(*=====================================================================*)
	IF 	Service.daten[i].Type_Service = STUNDEN THEN
		Service.visu[i].BtnType.Text := 'TIMER';
		Service.visu[i].BtnType.Pressed := FALSE;
	ELSIF 	Service.daten[i].Type_Service = TAGE THEN
		Service.visu[i].BtnType.Text := 'TIMER';
		Service.visu[i].BtnType.Pressed := FALSE;
	ELSIF Service.daten[i].Type_Service = COUNTER THEN
		Service.visu[i].BtnType.Text := 'COUNT';
		Service.visu[i].BtnType.Pressed := TRUE;
	END_IF
	Service.visu[i].BtnType.Enable := TRUE;
	Service.visu[i].BtnType.BackgroundColor := Color.lightgrey;
	Service.visu[i].BtnType.TextColor := Color.black;
	Service.visu[i].BtnType.Visible := TRUE;
END_FOR
END_ACTION
ACTION Reset:
k:=-1;
FOR k:=1 TO 3 BY 1 DO
	IF	gVarSystemtime.wHour >(MP.ShiftData.Shift[k].TimeStart.wHour + 1) AND NOT Reset_Help[k] THEN
		i:=-1;
		FOR i:=0 TO 15 BY 1 DO
			Default_reached[i] := FALSE;
		END_FOR
		Reset_Help[k]:=TRUE;
	END_IF
END_FOR

IF	gVarSystemtime.wHour < MP.ShiftData.Shift[1].TimeStart.wHour THEN
	k:=-1;
	FOR k:=1 TO 3 BY 1 DO
		Reset_Help[k]:=FALSE;
	END_FOR
END_IF
END_ACTION
ACTION Umschalten:
i := -1;

FOR i:=0 TO 15 BY 1 DO

(* Umschaltung der Funktion (Zeit oder Stückzahl) *)
	IF NOT b_first_cycle THEN
		IF	M_BtnType[i] AND NOT Service.visu[i].BtnType.Pressed THEN
				Service.daten[i].Starttag := 0;
				Service.daten[i].Startstunden := 0;
				Service.daten[i].StartBetriebsStd := 0;
				Service.daten[i].Current_Value := 0;
				IF	Service.daten[i].Type_Service < COUNTER THEN
						Service.daten[i].Type_Service:=Service.daten[i].Type_Service+1;
				ELSE
						Service.daten[i].Type_Service:=0;
				END_IF
		END_IF
		M_BtnType[i]:=Service.visu[i].BtnType.Pressed;

		IF	Service.daten[i].Type_Service = BETRIEBSSTUNDEN THEN
				Service.visu[i].BtnType.Text := 'TIMER';
				Service.daten[i].Unit := 'Betrieb Std';
		END_IF
		IF	Service.daten[i].Type_Service = STUNDEN THEN
				Service.visu[i].BtnType.Text := 'TIMER';
				Service.daten[i].Unit := 'Std';
		END_IF
		IF	Service.daten[i].Type_Service = TAGE THEN
				Service.visu[i].BtnType.Text := 'TIMER';
				Service.daten[i].Unit := 'Tage';
		END_IF
		IF	Service.daten[i].Type_Service = COUNTER THEN
				Service.visu[i].BtnType.Text := 'COUNT';
				Service.daten[i].Unit := 'Zähler';
		END_IF

	END_IF

	(*nur ganze Werte elauben*)
	IF	Service.daten[i].Type_Service = COUNTER OR
			Service.daten[i].Type_Service = TAGE THEN
			HelpString:=LREAL_TO_FMTSTR(Service.daten[i].Default_Value,0,TRUE);
			Service.daten[i].Default_Value:=STRING_TO_LREAL(HelpString);

			HelpString:=LREAL_TO_FMTSTR(Service.daten[i].Warning_Value,0,TRUE);
			Service.daten[i].Warning_Value:=STRING_TO_LREAL(HelpString);
	END_IF
	(* Werte auf 2 Stellen nach dem Komma begrenzen begrenzen*)
	IF	Service.daten[i].Type_Service = STUNDEN OR
			Service.daten[i].Type_Service = BETRIEBSSTUNDEN THEN
			HelpString:=LREAL_TO_FMTSTR(Service.daten[i].Default_Value,2,TRUE);
			Service.daten[i].Default_Value:=STRING_TO_LREAL(HelpString);

			HelpString:=LREAL_TO_FMTSTR(Service.daten[i].Warning_Value,2,TRUE);
			Service.daten[i].Warning_Value:=STRING_TO_LREAL(HelpString);
	END_IF

	(* aktuellen Werte löschen wenn Vorgabe und Warngrenze auf 0 steht*)
	IF	Service.daten[i].Warning_Value=0 AND Service.daten[i].Default_Value=0 THEN
			Service.daten[i].Current_Value:=0;
			Service.visu[i].Current_Value := '0';
			Service.daten[i].Starttag := 0;
			Service.daten[i].Startstunden := 0;
			Service.daten[i].StartBetriebsStd := 0;
			Service.daten[i].Current_Value := 0;
	END_IF

	(*======================================================================================================*)
	CASE Service.daten[i].Type_Service OF

	BETRIEBSSTUNDEN:
			(* Vorgabe erreicht Timer BETRIEBSSTUNDEN  *)
			IF	lr_Betriebsstunden - Service.daten[i].Default_Value >= Service.daten[i].StartBetriebsStd AND
					Service.daten[i].Default_Value >0 AND Service.daten[i].Startstunden >0 THEN
					Service.daten[i].Default_reached := TRUE;
			ELSE
					Service.daten[i].Default_reached := FALSE;
			END_IF

			(* Warngrenze erreicht Timer BETRIEBSSTUNDEN  *)
			IF	lr_Betriebsstunden - Service.daten[i].Warning_Value >= Service.daten[i].StartBetriebsStd AND
					Service.daten[i].Warning_Value >0 AND Service.daten[i].Startstunden >0 THEN
					Service.daten[i].Warning_reached := TRUE;
			ELSE
				Service.daten[i].Warning_reached := FALSE;
			END_IF

		(* Aktuellen Wert  auf der Visu anzeigen *)
		IF Service.daten[i].Starttag >0 THEN
			Service.visu[i].Current_Value :=LREAL_TO_FMTSTR(lr_Betriebsstunden - Service.daten[i].StartBetriebsStd,2,TRUE);
		ELSE
			Service.visu[i].Current_Value := '0';
		END_IF

		(* Start Button für BETRIEBSSTUNDEN sichtbar machen und bei betätigen den aktuellen Tag abspeichern *)
		IF 	Service.daten[i].Starttag =0 AND Service.daten[i].Default_Value >0 THEN
				Service.visu[i].BtnStart.Visible := TRUE;
				IF Service.visu[i].BtnStart.Pressed THEN
					Service.daten[i].Starttag := i_aktueller_tag;
					Service.daten[i].Startstunden := lr_aktuelle_stunden;
					Service.daten[i].StartBetriebsStd := lr_Betriebsstunden;
				END_IF
		ELSE
			Service.visu[i].BtnStart.Visible := FALSE;
		END_IF

	(*======================================================================================================*)
	STUNDEN:
			(* Vorgabe erreicht Timer STUNDEN  *)
			IF	(i_aktueller_tag * 24 + lr_aktuelle_stunden) - (Service.daten[i].Starttag * 24 + Service.daten[i].Startstunden) >= Service.daten[i].Default_Value AND
					Service.daten[i].Default_Value >0 AND Service.daten[i].Startstunden >0 THEN
					Service.daten[i].Default_reached := TRUE;
			ELSE
					Service.daten[i].Default_reached := FALSE;
			END_IF

			(* Warngrenze erreicht Timer STUNDEN  *)
			IF	(i_aktueller_tag * 24 + lr_aktuelle_stunden) - (Service.daten[i].Starttag * 24 + Service.daten[i].Startstunden) >= Service.daten[i].Warning_Value AND
					Service.daten[i].Warning_Value >0 AND Service.daten[i].Startstunden >0 THEN
					Service.daten[i].Warning_reached := TRUE;
			ELSE
				Service.daten[i].Warning_reached := FALSE;
			END_IF

		(* Aktuellen Wert  auf der Visu anzeigen *)
		IF Service.daten[i].Starttag >0 THEN
			Service.visu[i].Current_Value :=LREAL_TO_FMTSTR((i_aktueller_tag * 24 + lr_aktuelle_stunden) - (Service.daten[i].Starttag * 24 + Service.daten[i].Startstunden),2,TRUE);
		ELSE
			Service.visu[i].Current_Value := '0';
		END_IF

		(* Start Button für STUNDEN sichtbar machen und bei betätigen den aktuellen Tag abspeichern *)
		IF  Service.daten[i].Starttag =0 AND Service.daten[i].Default_Value >0 THEN
				Service.visu[i].BtnStart.Visible := TRUE;
				IF Service.visu[i].BtnStart.Pressed THEN
					Service.daten[i].Starttag := i_aktueller_tag;
					Service.daten[i].Startstunden := lr_aktuelle_stunden;
					Service.daten[i].StartBetriebsStd := lr_Betriebsstunden;
				END_IF
		ELSE
			Service.visu[i].BtnStart.Visible := FALSE;
		END_IF

	(*======================================================================================================*)
	TAGE:
		(* Vorgabe erreicht Timer TAGE*)
		IF (i_aktueller_tag - Service.daten[i].Starttag) >= Service.daten[i].Default_Value AND Service.daten[i].Default_Value >0 AND Service.daten[i].Starttag >0 THEN
			Service.daten[i].Default_reached := TRUE;
		ELSE
			Service.daten[i].Default_reached := FALSE;
		END_IF
		(* Warngrenze erreicht Timer TAGE  *)
		IF (i_aktueller_tag - Service.daten[i].Starttag) >= Service.daten[i].Warning_Value AND Service.daten[i].Warning_Value >0 AND Service.daten[i].Starttag >0 THEN
			Service.daten[i].Warning_reached := TRUE;
		ELSE
			Service.daten[i].Warning_reached := FALSE;
		END_IF

		(* Aktuellen Wert  auf der Visu anzeigen *)
		IF Service.daten[i].Starttag >0 THEN
			Service.visu[i].Current_Value := INT_TO_STRING (i_aktueller_tag - Service.daten[i].Starttag);
		ELSE
			Service.visu[i].Current_Value := '0';
		END_IF

		(* Start Button für TAGE sichtbar machen und bei betätigen den aktuellen Tag abspeichern *)
		IF  Service.daten[i].Starttag =0 AND Service.daten[i].Default_Value >0 THEN
				Service.visu[i].BtnStart.Visible := TRUE;
				IF Service.visu[i].BtnStart.Pressed THEN
					Service.daten[i].Starttag := i_aktueller_tag;
					Service.daten[i].Startstunden := lr_aktuelle_stunden;
					Service.daten[i].StartBetriebsStd := lr_Betriebsstunden;
				END_IF
		ELSE
			Service.visu[i].BtnStart.Visible := FALSE;
		END_IF

	(*======================================================================================================*)
	COUNTER:
	(* Vorgabe erreicht COUNTER*)
		IF Service.daten[i].Current_Value >= Service.daten[i].Default_Value AND Service.daten[i].Default_Value > 0 THEN
			Service.daten[i].Default_reached := TRUE;
		ELSE
			Service.daten[i].Default_reached := FALSE;
		END_IF
		(* Warngrenze erreicht COUNTER *)
		IF Service.daten[i].Current_Value >= Service.daten[i].Warning_Value AND Service.daten[i].Warning_Value > 0 THEN
			Service.daten[i].Warning_reached := TRUE;
		ELSE
			Service.daten[i].Warning_reached := FALSE;
		END_IF

	(* Aktuellen Wert  auf der Visu anzeigen *)
		Service.visu[i].Current_Value := LREAL_TO_FMTSTR(Service.daten[i].Current_Value, 0, TRUE);

		Service.visu[i].BtnStart.Visible := FALSE;
	END_CASE
	(*======================================================================================================*)

	(* Aktuellen Zähler reseten wenn dieser voll ist *)
	IF Service.daten[i].Default_reached OR Service.daten[i].Warning_reached THEN
		Service.visu[i].BtnReset.Visible := TRUE;	(* Den Resettaster nur anzeigen wenn Zähler>Vorgabe oder Zähler>Warnung *)
		IF Service.visu[i].BtnReset.Pressed THEN
			Service.daten[i].Starttag := 0;
			Service.daten[i].Startstunden := 0;
			Service.daten[i].StartBetriebsStd := 0;
			Service.daten[i].Current_Value := 0;
			Service.daten[i].Default_reached := FALSE;
			Service.daten[i].Warning_reached := FALSE;
			Default_reached[i]:=FALSE;
			Warning_reached[i]:=FALSE;
		END_IF
	ELSE
		Service.visu[i].BtnReset.Visible := FALSE;
	END_IF

	(* Farbwechsel des aktuellen Wertes *)
	IF Service.daten[i].Default_reached THEN
		Service.visu[i].Current_Value_Color := color.red;
	ELSIF Service.daten[i].Warning_reached AND NOT Service.daten[i].Default_reached THEN
		Service.visu[i].Current_Value_Color := color.yellow;
	ELSE
		Service.visu[i].Current_Value_Color := color.white;
	END_IF

END_FOR
END_ACTION

(* POU zLibrary/ept/Service/ST_BBGenXMLFile, ST *)
FUNCTION_BLOCK ST_BBGenXMLFile
VAR_INPUT
	(* ISK *)
	start_lesen_service						: BOOL;
	start_schreiben_service					: BOOL;

	(* Wo liegen die Dateien *)
	s_path								: STRING(255);

	(* Welche Dateien? *)
	s_service								: STRING(50);
END_VAR
VAR_OUTPUT
	fertig_lesen							: BOOL;
	fertig_schreiben						: BOOL;

	bError								: BOOL;
	nErrId								: UDINT;
END_VAR
VAR
	fb_state_entry							: ST_StateEntry;
	MsgOK								:BOOL;
	fb_ton_quitt							: TON;
	fb_xml_srv_write						: FB_XmlSrvWriteByName;
	fb_xml_srv_read						: FB_XmlSrvReadByName;
	s_file								: STRING(255);
	s_ErrorText							: STRING(255);
	ErrorID								:STRING(20);
END_VAR
fb_ton_quitt(IN:= , PT:= t#50ms, Q=> , ET=> );

(* ======================================Schrittkette======================================== *)
fb_state_entry(
	i16_next_step:= ,
	i16_pos:= 1,
	s_debugtext:= ,
	E=> ,
	X=> ,
	i16_step=> ,
	i16_last_step=> );


CASE fb_state_entry.i16_step OF
(*=======================================================*)
	0:
		bError := FALSE;
		nErrId := 0;

		s_file := '';
		s_ErrorText := '';
		fertig_lesen := FALSE;
		fertig_schreiben := FALSE;

	IF	fb_state_entry.fb_ton_Step.ET > t#10s THEN
		fb_state_entry.i16_next_step := 10;
	END_IF

(*=======================================================*)
	10:	(* Auslesen der Daten aus den XML-Files *)
		(* Daten lesen *)
		IF start_lesen_service THEN
			s_file := CONCAT(s_path, s_service);
			s_file := CONCAT(s_file,'.xml');
			fb_xml_srv_read.sSymName := '.service';
			fb_xml_srv_read.sXPath := '/root/service';
			fb_state_entry.i16_next_step := 100;
		END_IF

		(* Daten schreiben *)
		IF start_schreiben_service THEN
			s_file := CONCAT(s_path, s_service);
			s_file := CONCAT(s_file,'.xml');
			fb_xml_srv_write.sSymName := '.service';
			fb_xml_srv_write.sXPath := '/root/service';
			fb_state_entry.i16_next_step := 200;
		END_IF

(*=======================================================*)
	100:	(* Starte Daten lesen *)
		IF fb_state_entry.E THEN
			fb_xml_srv_read.bExecute := TRUE;
			fb_xml_srv_read.sFilePath := s_file;
		END_IF

		IF fb_xml_srv_read.bBusy THEN
			fb_xml_srv_read.bExecute := FALSE;
			fb_state_entry.i16_next_step := 110;
		END_IF

(*=======================================================*)
	110:	(* Lesevorgang *)
		IF NOT fb_xml_srv_read.bBusy  THEN
			IF NOT fb_xml_srv_read.bError THEN
				fb_state_entry.i16_next_step := 120;
			ELSE	(* Fehler *)
				nErrId := fb_xml_srv_read.nErrId;
				fb_state_entry.i16_next_step := 1000;
				ErrorID:='PM2';
				s_ErrorText:='Fehler beim Lesen der Service.xml Datei';
			END_IF
		END_IF

(*=======================================================*)
	120:	(* Lesevorgang beendet *)
		IF fb_state_entry.E THEN
			fertig_lesen := TRUE;
		END_IF

		IF NOT start_lesen_service THEN
			fb_state_entry.i16_next_step := 0;
		END_IF

(*=======================================================*)
	200:	(* Starte Daten schreiben *)
		IF fb_state_entry.E THEN
			fb_xml_srv_write.bExecute := TRUE;
			fb_xml_srv_write.sFilePath := s_file;
		END_IF

		IF fb_xml_srv_write.bBusy THEN
			fb_xml_srv_write.bExecute := FALSE;
			fb_state_entry.i16_next_step := 210;
		END_IF

(*=======================================================*)
	210:	(* Schreibvorgang *)
		IF NOT fb_xml_srv_write.bBusy  THEN
			IF NOT fb_xml_srv_write.bError THEN
				fb_state_entry.i16_next_step := 220;
			ELSE	(* Fehler *)
				nErrId := fb_xml_srv_write.nErrId;
				fb_state_entry.i16_next_step := 1000;
				s_ErrorText:=CONCAT('Fehler beim Schreiben der ',s_file);
			END_IF
		END_IF

(*=======================================================*)
	220:	(* Schreibvorgang beendet *)
		IF fb_state_entry.E THEN
			fertig_schreiben := TRUE;
		END_IF

		IF NOT start_schreiben_service THEN
			fb_state_entry.i16_next_step := 0;
		END_IF

(*=======================================================*)
	1000: (* Fehler *)
		IF fb_state_entry.E THEN
			MessageHandler.ClearMessageLines(sVisu:=Visu.Message);
		END_IF

		MessageHandler.Msg.ID:=ErrorID;
		MessageHandler.Msg.Color:=Color.red;
		MessageHandler.Msg.Name:='XML Error';
		MessageHandler.Msg.Text:=s_ErrorText;
		MessageHandler.Msg.Station:=0;

		MessageHandler(
			Prio:=2, 							(*1=highest, .. , 4=lowest*)
			Btn1Addr:=ADR(MsgOk),	(*Address of Button1 , if Zero then Button is unvisible*)
			Btn2Addr:=,						(*Address of Button2 , if Zero then Button is unvisible*)
			sVisu:=Visu.Message);

		(*-----------------------Weiterschaltbedingungen----------------------------*)
		IF MsgOK THEN
				MsgOk:=FALSE;
				fb_state_entry.i16_next_step:=0;
		END_IF

END_CASE


fb_state_entry(
	i16_next_step:= ,
	i16_pos:= 2,
	s_debugtext:= ,
	E=> , 
	X=> ,
	i16_step=> ,
	i16_last_step=> );

(* XML *)
fb_xml_srv_read(
	sNetId:= '',
	ePath:= PATH_GENERIC,
	nMode:= XMLSRV_SKIPMISSING,
	sSymName:= ,
	sFilePath:= ,
	sXPath:= ,
	bExecute:= ,
	tTimeout:= t#10s,
	bBusy=> ,
	bError=> ,
	nErrId=> );

fb_xml_srv_write(
	sNetId:= '',
	ePath:= PATH_GENERIC,
	nMode:= XMLSRV_ADDMISSING,
	sSymName:=  ,
	sFilePath:= ,
	sXPath:= ,
	bExecute:= ,
	tTimeout:= t#10s,
	bBusy=> ,
	bError=> ,
	nErrId=> );
END_FUNCTION_BLOCK

(* POU zLibrary/ept/Service/FB_Betriebsstundenzaehler, ST *)
FUNCTION_BLOCK FB_Betriebsstundenzaehler
VAR_INPUT
	Start					: BOOL;
	Reset					: BOOL;
	i32_betriebssekundenzaehler_in	: UDINT;
END_VAR
VAR_OUTPUT
	i32_betriebssekundenzaehler 	: UDINT;
	lr_betriebsstundenzaehler 		: LREAL;
END_VAR
VAR
	b_first_cycle					: BOOL := TRUE;
	fb_ton							: TON;
	t_betriebssekunden_Merker		: TIME := t#0ms;
	fb_r_trig_Reset					: R_TRIG;
	HelpString						: STRING(255);
END_VAR
IF b_first_cycle AND i32_betriebssekundenzaehler_in <>0 THEN
 	i32_betriebssekundenzaehler := i32_betriebssekundenzaehler_in;
	b_first_cycle := FALSE;
END_IF

fb_r_trig_Reset(CLK:=Reset , Q=> );
IF	fb_r_trig_Reset.Q THEN
		i32_betriebssekundenzaehler:=0;
END_IF

(* nach einer bestimmten Zeit speichern *)
IF	fb_ton.ET > t#15m THEN
		Start:=FALSE;
END_IF

IF NOT Start  THEN
	t_betriebssekunden_Merker := t_betriebssekunden_Merker + fb_ton.ET;
END_IF

fb_ton(IN:=Start, PT:= t#24h, Q=> , ET=> );

IF NOT Start THEN
	i32_betriebssekundenzaehler:=i32_betriebssekundenzaehler + (TIME_TO_UDINT(t_betriebssekunden_Merker)/1000);
	t_betriebssekunden_Merker:=t#0ms;
END_IF

lr_betriebsstundenzaehler:=UDINT_TO_LREAL(i32_betriebssekundenzaehler) / 3600;
HelpString:=LREAL_TO_FMTSTR(lr_betriebsstundenzaehler,2,TRUE);
lr_betriebsstundenzaehler:=STRING_TO_LREAL(HelpString);
END_FUNCTION_BLOCK

(* POU Stations/ST_00/ST00_PRGs/ST00_ImpExp_MP, ST *)
PROGRAM ST00_ImpExp_MP
VAR_INPUT
	Start_write				:BOOL;
	Start_read				:BOOL;
	path						:STRING(255);
	filename					:STRING(255);
END_VAR
VAR
	b_init					:BOOL;
	fb_state_entry				:ST_StateEntry;

	fb_xml_srv_read			: FB_XmlSrvReadByName;
	fb_xml_srv_write			: FB_XmlSrvWriteByName;

	fb_rtrig_Start_read			:R_TRIG;
	fb_rtrig_Start_write_to_server:R_TRIG;
	fb_ton_init				:TON;
	fb_ton_wz				:TON;
	fb_ton_uez				:TON;

	bError					: BOOL;
	nErrId					: UDINT;
	s_info					: STRING;
	MsgOK					: BOOL;
	MsgID					:STRING(20);
	MP_Copy				: sMachPara;
END_VAR

VAR_OUTPUT
	Busy					:BOOL;
	Done					:BOOL;
	Error					:BOOL;
	ErrorMsg					:STRING(255);
END_VAR

VAR CONSTANT
	SymName				:STRING:='.MP';
	xPath					:STRING:='/MP';
END_VAR

VAR_IN_OUT

END_VAR
(*======================================================
   PRG: XML Import und Export der MD
 ------------------------------------------------------
   Auth: 		Werner Friedl    						 
   Date: 		25.10.2017   						     
   Rev.: 		1.0	
   Desc:		
	- Maschinen Parameter werden beim Neustart eingelesen
	- bei einer Änderung wird die Änderung automatisch in die xml eingeragen

   Historie:   1.0



 ========================================================*)
fb_ton_init(IN:= TRUE, PT:=t#1500ms , Q=> , ET=> );
IF	NOT b_init AND fb_ton_init.Q THEN
	Start_read := TRUE;
	b_Init:=TRUE;
END_IF

(* ========================================================*)
fb_rtrig_Start_read();
IF	fb_rtrig_Start_read.Q AND
	NOT Start_write THEN
	Start_read:=TRUE;
END_IF

IF 	(MEMCMP(ADR(MP_Copy),ADR(MP),SIZEOF(MP_Copy))<>0)AND (*automatisch speichern im Manualmode*)
     	ModeSelect.Mode <=MODE_MANUAL AND
	NOT Start_read AND
	b_Init THEN
	Start_write := TRUE;
END_IF

(* ========================================================*)
fb_ton_wz(IN:= , PT:=t#3000ms , Q=> , ET=> );
IF	fb_ton_wz.Q THEN
	fb_ton_wz.IN:=FALSE;
	s_info := '';
END_IF

fb_state_entry(i16_pos:= 1);
CASE fb_state_entry.i16_step OF

(*=======================================================*)
INIT_OBJ:
	fb_state_entry.i16_next_step:=INIT;

(*=======================================================*)
INIT: fb_state_entry.s_debugtext:='initialisieren';

	Start_write := FALSE;
	Start_read := FALSE;
	fb_state_entry.i16_next_step:=BEREIT;

(*=======================================================*)
BEREIT:fb_state_entry.s_debugtext:='warte auf start';

	IF	Start_read THEN
		fb_state_entry.i16_next_step:=110;
	END_IF

	IF	Start_write THEN
		fb_state_entry.i16_next_step:=200;
	END_IF

	IF fb_state_entry.X THEN
		fb_ton_uez.IN:=FALSE;
		Start_write:=FALSE;
		Start_read:=FALSE;
		Busy:=TRUE;
		Error:=FALSE;
		Done:=FALSE;
		nErrId:=0;
		ErrorMsg:='';
		MsgID:='';
	END_IF

(*=======================================================*)
110: fb_state_entry.s_debugtext:='XML auslesen';

	IF fb_state_entry.E THEN
		(*MD:=MD_leer;*)
		fb_xml_srv_read.sFilePath := CONCAT(path,filename);
		fb_xml_srv_read.sSymName:=SymName;
		fb_xml_srv_read.sXPath :=xPath;
		fb_xml_srv_read.bExecute := TRUE;
	END_IF

	IF fb_xml_srv_read.bBusy THEN
		fb_xml_srv_read.bExecute := FALSE;
		fb_state_entry.i16_next_step := 120;
	END_IF

(*=======================================================*)
120:fb_state_entry.s_debugtext:='Lesevorgang erfolgreich?';

	IF  NOT fb_xml_srv_read.bBusy  THEN
		IF NOT fb_xml_srv_read.bError THEN
			fb_state_entry.i16_next_step := 900;
		ELSE	(* Fehler *)
			nErrId := fb_xml_srv_read.nErrId;
			IF	nErrId =1804 THEN
				MsgID:='PM5';
				ErrorMsg:='Die Datei MP.xml ist nicht vorhanden';
				fb_state_entry.i16_next_step := 200;	(*Datei wird erstellt*)
			ELSE
				MsgID:='PM6';
				ErrorMsg:='Fehler beim Einlesen der MP.xml Datei';
				fb_state_entry.i16_next_step := FEHLER;
			END_IF
		END_IF
	END_IF

	IF fb_state_entry.X THEN
		fb_ton_wz.IN:=TRUE;
		s_info:=CONCAT('read ',filename);
	END_IF

(*=======================================================*)
200:fb_state_entry.s_debugtext:='XML schreiben';

	IF fb_state_entry.E THEN
		fb_xml_srv_write.sFilePath := CONCAT(path,filename);
		fb_xml_srv_write.sSymName:=SymName;
		fb_xml_srv_write.sXPath :=xPath;
		fb_xml_srv_write.bExecute := TRUE;
	END_IF

	IF fb_xml_srv_write.bBusy THEN
		fb_xml_srv_write.bExecute := FALSE;
		fb_state_entry.i16_next_step := 220;
	END_IF

(*=======================================================*)
220:fb_state_entry.s_debugtext:='Schreiben erfolgreich?';

	IF  NOT fb_xml_srv_write.bBusy  THEN
		IF NOT fb_xml_srv_write.bError THEN
			MP_Copy := MP;
			fb_state_entry.i16_next_step := 900;
		ELSE	(* Fehler *)
			nErrId := fb_xml_srv_write.nErrId;
			MsgID:='PM7';
			ErrorMsg:='Fehler beim Schreiben der MP.xml';
			fb_state_entry.i16_next_step := FEHLER;
		END_IF
	END_IF

	IF fb_state_entry.X THEN
		fb_ton_wz.IN:=TRUE;
		fb_ton_uez.IN:=TRUE;		(*automatisch auf Server speichern*)
		s_info:=CONCAT('write ',filename);
	END_IF

(*=======================================================*)
900:fb_state_entry.s_debugtext:='Fertig';

	Busy:=FALSE;
	Done:=TRUE;
	fb_state_entry.i16_next_step:=0;

(*=======================================================*)
FEHLER:

	IF fb_state_entry.E THEN
		MessageHandler.ClearMessageLines(sVisu:=Visu.Message);
	END_IF
	MessageHandler.Msg.ID:=MsgID;
	MessageHandler.Msg.Name:=ErrorMsg;
	MessageHandler.Msg.Text:=ErrorMsg;
	MessageHandler.Msg.Color:=Color.red;
	MessageHandler.Msg.Station:=0;

	MessageHandler(
		Prio:=2, 							(*1=highest, .. , 4=lowest*)
		Btn1Addr:=ADR(MsgOk),			(*Address of Button1 , if Zero then Button is unvisible*)
		Btn2Addr:=,						(*Address of Button2 , if Zero then Button is unvisible*)
		sVisu:=Visu.Message);

	IF MsgOK THEN
		MsgOk:=FALSE;
		fb_state_entry.i16_next_step:=0;
		Busy:=FALSE;
		Error:=TRUE;
	END_IF
END_CASE

fb_state_entry(i16_pos:= 2);


fb_xml_srv_read(
	sNetId:= '',
	ePath:= PATH_GENERIC,
	nMode:= XMLSRV_SKIPMISSING,
	sSymName:= ,
	sFilePath:= ,
	sXPath:= ,
	bExecute:= ,
	tTimeout:= t#10s,
	bBusy=> ,
	bError=> ,
	nErrId=> );

fb_xml_srv_write(
	sNetId:= '',
	ePath:= PATH_GENERIC,
	nMode:= XMLSRV_ADDMISSING,
	sSymName:=  ,
	sFilePath:= ,
	sXPath:= ,
	bExecute:= ,
	tTimeout:= t#10s,
	bBusy=> ,
	bError=> ,
	nErrId=> );


(*automatisch auf Server speichern=============================================*)
fb_ton_uez(PT:=t#20s);
fb_rtrig_Start_write_to_server(CLK:=fb_ton_uez.Q , Q=> );
(*
NT_StartProcess(
	NETID:='',
	PATHSTR	:='C:\Windows\System32\cmd.exe',
	DIRNAME	:='D:\Tools ',
	COMNDLINE	:='/C copy C:\MP\MachPara.xml \\10.16.50.9\bbgen\UML3\MD & @ping localhost -n 4 >NUL',
	START		:=fb_rtrig_Start_write_to_server.Q,
	TMOUT		:=t#10s);
*)
(*
NT_StartProcess(
	NETID:='',
	PATHSTR	:='C:\Windows\System32\wscript.exe',
	DIRNAME	:='D:\Tools',
	COMNDLINE	:='de_PD_aktuell_von_uml_nach_server.vbs',
	START		:=fb_rtrig_Start_write_to_server.Q,
	TMOUT		:=t#10s);
*)
END_PROGRAM

(* POU Stations/ST_02_RT_Tampondrucker/ST02_PRGs/ST02_CallPRGs, ST *)
PROGRAM ST02_CallPRGs

VAR
	FB_ReadXmlLineConf		: FB_ReadXmlLine;
	sDescription			: STRING;
END_VAR
TurnTable();

IF 	ST02_HomePosition.State = STATE_RUN THEN
	ListHomeNOK(InstName:='ST02 ',Description:=sDescription);
END_IF
FB_ReadXmlLineConf(
	Prefix:= 'CONFIG',
	ID:= 'ST02',
	File:= 'CONFIG.xml',
	Text=> sDescription );

(*Hauptluft Tampondrucker einschalten*)
IF 	ST08_210_S2.BitInToCheck THEN	(*   Not-Aus 2 TD ausgelöst (DigIn) *)
	ST02_35Y01.MoveWork:=TRUE;
ELSE
	ST02_35Y01.MoveInit:=TRUE;
END_IF
END_PROGRAM

(* POU Stations/ST_02_RT_Tampondrucker/ST02_PRGs/TurnTable, ST *)
PROGRAM TurnTable
VAR_OUTPUT
	TurnEnable				: BOOL;
	TurnDisableString		: STRING(255);
END_VAR
VAR
	Test					: BOOL;
	TurnImp					: R_TRIG;

	TimeOutError			: BOOL;
	NestIdx					: DINT;
END_VAR
(*Interlocking for Turn-Table (used in Manual- and in AutoMode)
  ----------------------------------------------------------------------------------------*)

IF 	Robot01.ActualArea=3 THEN	(*Belade-Roboter bei Rundtisch*)
	TurnEnable:=FALSE;
	TurnDisableString:='Robot01.ActualArea=3 in Rundtisch';
ELSIF
	TimeOutError THEN			(*TimeOutError*)
	TurnEnable:=FALSE;
	TurnDisableString:='TimeOutError';
ELSIF
	ST00_220_S1.BitInToCheck THEN (* Schutz nicht geschlossen*)
	TurnEnable:=FALSE;
	TurnDisableString:='Schutztüre nicht geschlossen! ()';
ELSE
	TurnEnable:=TRUE;
	TurnDisableString:='';
END_IF

(*Daten schieben, wenn Rundtisch dreht
	  ----------------------------------------------------------------------------------------*)
IF ModeSelect.Mode=MODE_MANUAL THEN
	TurnImp(CLK:=		(*ST02_162_A1_3.BitOutToSet OR *)  (*Drehen*)
				Test);
	IF TurnImp.Q THEN
		MP.ST02.TableData:=PushData(MP.ST02.TableData);
	END_IF
END_IF
(*Calculate Table Empty*)
gTableEmpty:=TRUE;
FOR NestIdx:=1 TO NO_OF_NEST DO
	IF 	MP.ST02.TableData[NestIdx].ProcessData.Part THEN
		gTableEmpty:=FALSE;
		EXIT;
	END_IF
END_FOR
END_PROGRAM

(* POU Stations/ST_03_Ruestsaetze/ST_03_PRGs/ST03_CallPRGs, ST *)
PROGRAM ST03_CallPRGs
VAR
	fbTon_EndTestParts    	: TON;
	fb_rTrig_EndTestParts	: R_TRIG;
	fb_rTrig_TestParts 		: R_TRIG;

	FB_ReadXmlLineConf		: FB_ReadXmlLine;
	sDescription			: STRING;
	i						:INT;
 	ST03_Ruestsatz			: ARRAY[1..3] OF SFCCurrent;	(*für Grundstellungs Info*)
 	ST03_RuestsatzEmpty		: ARRAY[1..3] OF SFCCurrent;

END_VAR
ST03_ManRobotSwivelUnit();
ST03_Band();
ST03_Test_Parts();
ST03_Init_Lockings();
ST03_Init_AbholPos();

IF 	ST02_HomePosition.State = STATE_RUN THEN
	ListHomeNOK(InstName:='ST03 ',Description:=sDescription);
END_IF

FB_ReadXmlLineConf(
	Prefix:= 'CONFIG',
	ID:= 'ST03',
	File:= 'CONFIG.xml',
	Text=> sDescription );

(*Clear GipperState, if Gripper is opened*)
IF	 Robot01.RemInToolWorkSensor THEN
	gRob01GripState:=PART_NO;
END_IF

ST03_Autostop();

MP.ST03.NoOfTestParts:=MP.ST03.NoOfTestParts - (MP.ST03.NoOfTestParts MOD TD.PartsInRoboGripper);
IF 	MP.ST03.NoOfTestParts < TD.PartsInRoboGripper THEN
	MP.ST03.NoOfTestParts:=TD.PartsInRoboGripper;
END_IF

(* Förderband Prüfteile *)
IF 	MP.ST03.BeltMotorCheckPartActive THEN
	fbTon_EndTestParts(IN:=NOT gTakeTestParts,PT:=t#10s);
	fb_rTrig_TestParts(CLK:=
						gTakeTestParts AND
						ModeSelect.Mode>MODE_MANUAL);
	fb_rTrig_EndTestParts(CLK:=
						fbTon_EndTestParts.Q OR
						ModeSelect.Mode=MODE_MANUAL);

	IF 	fb_rTrig_TestParts.Q THEN
		ST03_601V1_A1.SetSignalHigh:=TRUE;
	END_IF
	IF	fb_rTrig_EndTestParts.Q THEN
    	ST03_601V1_A1.SetSignalLow:=TRUE;
	END_IF

END_IF
(* Berechnung aller Schlechtteile*)
i32_total_NOK_parts :=gNokPartsColorCam+gNokPartsWingCam+i32_first_parts;

(*Hauptluft Tintenstrahldrucker einschalten nur bei SG-Maschine 3621*)
IF 	MP.ST03.SGM_3621 THEN
	IF 	ST08_210_S2.BitInToCheck THEN	(*   Not-Aus 2 TD ausgelöst (DigIn) *)
		ST03_Y01.MoveWork:=TRUE;
	ELSE
		ST03_Y01.MoveInit:=TRUE;
	END_IF
END_IF

ST03_Ruestsatz:=ST03_RuestsatzEmpty;

CASE  gTypeCode OF
(*160pol============================================================================*)
322:
	ST03_160pol_Zufuehrung(
		b_Printer_Off:=TRUE,
		SFCCurrentPOU=> ST03_Ruestsatz[1].SFCCurrentPOU,
		SFCCurrentStep=> ST03_Ruestsatz[1].SFCCurrentStep,
		SFCTime=>ST03_Ruestsatz[1].SFCTime );
	ST03_160pol_Zufuehrung.FB_CurrentStepHistorie(st_CurrentStep:=ST03_160pol_Zufuehrung.SFCCurrentStep);

	IF	(ModeSelect.Mode=MODE_AUTO_RUN OR 	ModeSelect.Mode=MODE_STEP_RUN) AND
		NOT gRunEmpty THEN
		ST03_160pol_Zufuehrung.Start:=TRUE;
	ELSE
		ST03_160pol_Zufuehrung.Start:=FALSE;
	END_IF

(*154pol=============================================================================*)
4871:
	ST03_154pol_Zufuehrung(
		SFCCurrentPOU=> ST03_Ruestsatz[1].SFCCurrentPOU,
		SFCCurrentStep=> ST03_Ruestsatz[1].SFCCurrentStep,
		SFCTime=>ST03_Ruestsatz[1].SFCTime );
	ST03_154pol_Zufuehrung.FB_CurrentStepHistorie(st_CurrentStep:=ST03_154pol_Zufuehrung.SFCCurrentStep);

	IF	(ModeSelect.Mode=MODE_AUTO_RUN OR 	ModeSelect.Mode=MODE_STEP_RUN)	AND
		NOT gRunEmpty THEN
		ST03_154pol_Zufuehrung.Start:=TRUE;
	ELSE
		ST03_154pol_Zufuehrung.Start:=FALSE;
	END_IF

(*154 Rasterplatte=============================================================================*)
4872:
	ST03_154_RP_Zufuehrung(
		SFCCurrentPOU=> ST03_Ruestsatz[1].SFCCurrentPOU,
		SFCCurrentStep=> ST03_Ruestsatz[1].SFCCurrentStep,
		SFCTime=>ST03_Ruestsatz[1].SFCTime );
	ST03_154_RP_Zufuehrung.FB_CurrentStepHistorie(st_CurrentStep:=ST03_154_RP_Zufuehrung.SFCCurrentStep);

	IF	(ModeSelect.Mode=MODE_AUTO_RUN OR 	ModeSelect.Mode=MODE_STEP_RUN)	AND
		NOT gRunEmpty THEN
		ST03_154_RP_Zufuehrung.Start:=TRUE;
	ELSE
		ST03_154_RP_Zufuehrung.Start:=FALSE;
	END_IF

(*93pol, 102pol=============================================================================*)
312,4991:
	ST03_102pol_Zufuehrung(
		SFCCurrentPOU=> ST03_Ruestsatz[1].SFCCurrentPOU,
		SFCCurrentStep=> ST03_Ruestsatz[1].SFCCurrentStep,
		SFCTime=>ST03_Ruestsatz[1].SFCTime );
	ST03_102pol_Zufuehrung.FB_CurrentStepHistorie(st_CurrentStep:=ST03_102pol_Zufuehrung.SFCCurrentStep);

	IF	(ModeSelect.Mode=MODE_AUTO_RUN OR 	ModeSelect.Mode=MODE_STEP_RUN)OR MP.ST02.DummyPruefung_93pol	AND
		NOT gRunEmpty THEN
		ST03_102pol_Zufuehrung.Start:=TRUE;
	ELSE
		ST03_102pol_Zufuehrung.Start:=FALSE;
	END_IF
	IF	MP.ST00.IFMCameraActive THEN
		ST03_IFM_Camera();
		ST03_IFM_Camera.FB_CurrentStepHistorie(st_CurrentStep:=ST03_IFM_Camera.SFCCurrentStep);
	END_IF

(*206pol=============================================================================*)
522:
	ST03_206pol_Zufuehrung(
		SFCCurrentPOU=> ST03_Ruestsatz[1].SFCCurrentPOU,
		SFCCurrentStep=> ST03_Ruestsatz[1].SFCCurrentStep,
		SFCTime=>ST03_Ruestsatz[1].SFCTime );
	ST03_206pol_Zufuehrung.FB_CurrentStepHistorie(st_CurrentStep:=ST03_206pol_Zufuehrung.SFCCurrentStep);

	IF	(ModeSelect.Mode=MODE_AUTO_RUN OR 	ModeSelect.Mode=MODE_STEP_RUN)	AND
		NOT gRunEmpty THEN
		ST03_206pol_Zufuehrung.Start:=TRUE;
	ELSE
		ST03_206pol_Zufuehrung.Start:=FALSE;
	END_IF

(*92pol=============================================================================*)
550:
	ST03_92pol_Zufuehrung(
		SFCCurrentPOU=> ST03_Ruestsatz[1].SFCCurrentPOU,
		SFCCurrentStep=> ST03_Ruestsatz[1].SFCCurrentStep,
		SFCTime=>ST03_Ruestsatz[1].SFCTime );
	ST03_92pol_Zufuehrung.FB_CurrentStepHistorie(st_CurrentStep:=ST03_92pol_Zufuehrung.SFCCurrentStep);

	IF	(ModeSelect.Mode=MODE_AUTO_RUN OR 	ModeSelect.Mode=MODE_STEP_RUN)	AND
		NOT gRunEmpty THEN
		ST03_92pol_Zufuehrung.Start:=TRUE;
	ELSE
		ST03_92pol_Zufuehrung.Start:=FALSE;
	END_IF

(*124pol=============================================================================*)
564:
	ST03_124pol_Zufuehrung(
		SFCCurrentPOU=> ST03_Ruestsatz[1].SFCCurrentPOU,
		SFCCurrentStep=> ST03_Ruestsatz[1].SFCCurrentStep,
		SFCTime=>ST03_Ruestsatz[1].SFCTime );
	ST03_124pol_Zufuehrung.FB_CurrentStepHistorie(st_CurrentStep:=ST03_124pol_Zufuehrung.SFCCurrentStep);

	IF	(ModeSelect.Mode=MODE_AUTO_RUN OR 	ModeSelect.Mode=MODE_STEP_RUN)	AND
		NOT gRunEmpty THEN
		ST03_124pol_Zufuehrung.Start:=TRUE;
	ELSE
		ST03_124pol_Zufuehrung.Start:=FALSE;
	END_IF

(*46pol=============================================================================*)
569:
	ST03_46pol_Zufuehrung(
		SFCCurrentPOU=> ST03_Ruestsatz[1].SFCCurrentPOU,
		SFCCurrentStep=> ST03_Ruestsatz[1].SFCCurrentStep,
		SFCTime=>ST03_Ruestsatz[1].SFCTime );
	ST03_46pol_Zufuehrung.FB_CurrentStepHistorie(st_CurrentStep:=ST03_46pol_Zufuehrung.SFCCurrentStep);
	ST03_46pol_Wendeeinheit(
		SFCCurrentPOU=> ST03_Ruestsatz[2].SFCCurrentPOU,
		SFCCurrentStep=> ST03_Ruestsatz[2].SFCCurrentStep,
		SFCTime=>ST03_Ruestsatz[2].SFCTime );
	ST03_46pol_Wendeeinheit.FB_CurrentStepHistorie(st_CurrentStep:=ST03_46pol_Wendeeinheit.SFCCurrentStep);


	IF	(ModeSelect.Mode=MODE_AUTO_RUN OR 	ModeSelect.Mode=MODE_STEP_RUN)	AND
		NOT gRunEmpty THEN
		ST03_46pol_Zufuehrung.Start:=TRUE;
		ST03_46pol_Wendeeinheit.Start:=TRUE;
	ELSE
		ST03_46pol_Zufuehrung.Start:=FALSE;
		ST03_46pol_Wendeeinheit.Start:=FALSE;
	END_IF

(*NOX 4pol=============================================================================*)
5631:
	ST03_NOX_4pol_Zufuehrung(
		SFCCurrentPOU=> ST03_Ruestsatz[1].SFCCurrentPOU,
		SFCCurrentStep=> ST03_Ruestsatz[1].SFCCurrentStep,
		SFCTime=>ST03_Ruestsatz[1].SFCTime );
	ST03_NOX_4pol_Zufuehrung.FB_CurrentStepHistorie(st_CurrentStep:=ST03_NOX_4pol_Zufuehrung.SFCCurrentStep);

	IF	(ModeSelect.Mode=MODE_AUTO_RUN OR 	ModeSelect.Mode=MODE_STEP_RUN)	AND
		NOT gRunEmpty THEN
		ST03_NOX_4pol_Zufuehrung.Start:=TRUE;
		ST03_65_Q1.SetSignalHigh := TRUE;		(*Kühltunnel (Lüfter)*)
	ELSE
		ST03_NOX_4pol_Zufuehrung.Start:=FALSE;
		ST03_65_Q1.SetSignalLow := TRUE;		(*Kühltunnel (Lüfter)*)
	END_IF

(*NOX 5pol=============================================================================*)
5632:
	ST03_NOX_5pol_Zufuehrung(
		SFCCurrentPOU=> ST03_Ruestsatz[1].SFCCurrentPOU,
		SFCCurrentStep=> ST03_Ruestsatz[1].SFCCurrentStep,
		SFCTime=>ST03_Ruestsatz[1].SFCTime );
	ST03_NOX_5pol_Zufuehrung.FB_CurrentStepHistorie(st_CurrentStep:=ST03_NOX_5pol_Zufuehrung.SFCCurrentStep);

	IF	(ModeSelect.Mode=MODE_AUTO_RUN OR 	ModeSelect.Mode=MODE_STEP_RUN)	AND
		NOT gRunEmpty THEN
		ST03_NOX_5pol_Zufuehrung.Start:=TRUE;
		ST03_65_Q1.SetSignalHigh := TRUE;		(*Kühltunnel (Lüfter)*)
	ELSE
		ST03_NOX_5pol_Zufuehrung.Start:=FALSE;
		ST03_65_Q1.SetSignalLow := TRUE;		(*Kühltunnel (Lüfter)*)
	END_IF

(*NOX 6pol=============================================================================*)
5633:
	ST03_NOX_6pol_Zufuehrung(
		SFCCurrentPOU=> ST03_Ruestsatz[1].SFCCurrentPOU,
		SFCCurrentStep=> ST03_Ruestsatz[1].SFCCurrentStep,
		SFCTime=>ST03_Ruestsatz[1].SFCTime );
	ST03_NOX_6pol_Zufuehrung.FB_CurrentStepHistorie(st_CurrentStep:=ST03_NOX_6pol_Zufuehrung.SFCCurrentStep);

	IF	(ModeSelect.Mode=MODE_AUTO_RUN OR 	ModeSelect.Mode=MODE_STEP_RUN)	AND
		NOT gRunEmpty THEN
		ST03_NOX_6pol_Zufuehrung.Start:=TRUE;
		ST03_65_Q1.SetSignalHigh := TRUE;		(*Kühltunnel (Lüfter)*)
	ELSE
		ST03_NOX_6pol_Zufuehrung.Start:=FALSE;
		ST03_65_Q1.SetSignalLow := TRUE;		(*Kühltunnel (Lüfter)*)
	END_IF

(*88pol=============================================================================*)
5731:
	ST03_88pol_Zufuehrung(
		SFCCurrentPOU=> ST03_Ruestsatz[1].SFCCurrentPOU,
		SFCCurrentStep=> ST03_Ruestsatz[1].SFCCurrentStep,
		SFCTime=>ST03_Ruestsatz[1].SFCTime );
	ST03_88pol_Zufuehrung.FB_CurrentStepHistorie(st_CurrentStep:=ST03_88pol_Zufuehrung.SFCCurrentStep);

	IF	(ModeSelect.Mode=MODE_AUTO_RUN OR 	ModeSelect.Mode=MODE_STEP_RUN)	AND
		NOT gRunEmpty THEN
		ST03_88pol_Zufuehrung.Start:=TRUE;
	ELSE
		ST03_88pol_Zufuehrung.Start:=FALSE;
	END_IF

(*7pol=============================================================================*)
575,5753,5754:
	ST03_7pol_Zufuehrung(
		SFCCurrentPOU=> ST03_Ruestsatz[1].SFCCurrentPOU,
		SFCCurrentStep=> ST03_Ruestsatz[1].SFCCurrentStep,
		SFCTime=>ST03_Ruestsatz[1].SFCTime );
	ST03_7pol_Zufuehrung.FB_CurrentStepHistorie(st_CurrentStep:=ST03_7pol_Zufuehrung.SFCCurrentStep);
	ST03_7pol_Wendeeinheit(
		SFCCurrentPOU=> ST03_Ruestsatz[2].SFCCurrentPOU,
		SFCCurrentStep=> ST03_Ruestsatz[2].SFCCurrentStep,
		SFCTime=>ST03_Ruestsatz[2].SFCTime );
	ST03_7pol_Wendeeinheit.FB_CurrentStepHistorie(st_CurrentStep:=ST03_7pol_Wendeeinheit.SFCCurrentStep);
	IF	(ModeSelect.Mode=MODE_AUTO_RUN OR 	ModeSelect.Mode=MODE_STEP_RUN)	AND
		NOT gRunEmpty THEN
		ST03_7pol_Zufuehrung.Start:=TRUE;
		ST03_7pol_Wendeeinheit.Start:=TRUE;
	ELSE
		ST03_7pol_Zufuehrung.Start:=FALSE;
		ST03_7pol_Wendeeinheit.Start:=FALSE;
	END_IF

(*9pol=============================================================================*)
5755:
	ST03_7pol_Zufuehrung(
		SFCCurrentPOU=> ST03_Ruestsatz[1].SFCCurrentPOU,
		SFCCurrentStep=> ST03_Ruestsatz[1].SFCCurrentStep,
		SFCTime=>ST03_Ruestsatz[1].SFCTime );
	ST03_7pol_Zufuehrung.FB_CurrentStepHistorie(st_CurrentStep:=ST03_7pol_Zufuehrung.SFCCurrentStep);
	ST03_9pol_Wendeeinheit(
		SFCCurrentPOU=> ST03_Ruestsatz[2].SFCCurrentPOU,
		SFCCurrentStep=> ST03_Ruestsatz[2].SFCCurrentStep,
		SFCTime=>ST03_Ruestsatz[2].SFCTime );
	ST03_9pol_Wendeeinheit.FB_CurrentStepHistorie(st_CurrentStep:=ST03_7pol_Wendeeinheit.SFCCurrentStep);
	IF	(ModeSelect.Mode=MODE_AUTO_RUN OR 	ModeSelect.Mode=MODE_STEP_RUN)	AND
		NOT gRunEmpty THEN
		ST03_7pol_Zufuehrung.Start:=TRUE;
		ST03_9pol_Wendeeinheit.Start:=TRUE;
	ELSE
		ST03_7pol_Zufuehrung.Start:=FALSE;
		ST03_9pol_Wendeeinheit.Start:=FALSE;
	END_IF

(*88pol AMG=============================================================================*)
5732:
	ST03_88polAMG_Zufuehrung(
		SFCCurrentPOU=> ST03_Ruestsatz[1].SFCCurrentPOU,
		SFCCurrentStep=> ST03_Ruestsatz[1].SFCCurrentStep,
		SFCTime=>ST03_Ruestsatz[1].SFCTime );
	ST03_88polAMG_Zufuehrung.FB_CurrentStepHistorie(st_CurrentStep:=ST03_88polAMG_Zufuehrung.SFCCurrentStep);

	IF	(ModeSelect.Mode=MODE_AUTO_RUN OR 	ModeSelect.Mode=MODE_STEP_RUN)	AND
		NOT gRunEmpty THEN
		ST03_88polAMG_Zufuehrung.Start:=TRUE;
	ELSE
		ST03_88polAMG_Zufuehrung.Start:=FALSE;
	END_IF

(*120pol AMG=============================================================================*)
5771:
	ST03_120pol_Zufuehrung(
		SFCCurrentPOU=> ST03_Ruestsatz[1].SFCCurrentPOU,
		SFCCurrentStep=> ST03_Ruestsatz[1].SFCCurrentStep,
		SFCTime=>ST03_Ruestsatz[1].SFCTime );
	ST03_120pol_Zufuehrung.FB_CurrentStepHistorie(st_CurrentStep:=ST03_120pol_Zufuehrung.SFCCurrentStep);

	IF	(ModeSelect.Mode=MODE_AUTO_RUN OR 	ModeSelect.Mode=MODE_STEP_RUN)	AND
		NOT gRunEmpty THEN
		ST03_120pol_Zufuehrung.Start:=TRUE;
	ELSE
		ST03_120pol_Zufuehrung.Start:=FALSE;
	END_IF


(*21pol AMG=============================================================================*)
5772:
	ST03_21pol_Zufuehrung(
		SFCCurrentPOU=> ST03_Ruestsatz[1].SFCCurrentPOU,
		SFCCurrentStep=> ST03_Ruestsatz[1].SFCCurrentStep,
		SFCTime=>ST03_Ruestsatz[1].SFCTime );
	ST03_21pol_Zufuehrung.FB_CurrentStepHistorie(st_CurrentStep:=ST03_21pol_Zufuehrung.SFCCurrentStep);

	IF	(ModeSelect.Mode=MODE_AUTO_RUN OR 	ModeSelect.Mode=MODE_STEP_RUN)	AND
		NOT gRunEmpty THEN
		ST03_21pol_Zufuehrung.Start:=TRUE;
	ELSE
		ST03_21pol_Zufuehrung.Start:=FALSE;
	END_IF

(*191pol =============================================================================*)
580:
	ST03_191pol_Zufuehrung(
		SFCCurrentPOU=> ST03_Ruestsatz[1].SFCCurrentPOU,
		SFCCurrentStep=> ST03_Ruestsatz[1].SFCCurrentStep,
		SFCTime=>ST03_Ruestsatz[1].SFCTime );
	ST03_191pol_Zufuehrung.FB_CurrentStepHistorie(st_CurrentStep:=ST03_191pol_Zufuehrung.SFCCurrentStep);

	IF	(ModeSelect.Mode=MODE_AUTO_RUN OR 	ModeSelect.Mode=MODE_STEP_RUN)	AND
		NOT gRunEmpty THEN
		ST03_191pol_Zufuehrung.Start:=TRUE;
	ELSE
		ST03_191pol_Zufuehrung.Start:=FALSE;
	END_IF

(*72pol =============================================================================*)
5831:
	ST03_72pol_Zufuehrung(
		SFCCurrentPOU=> ST03_Ruestsatz[1].SFCCurrentPOU,
		SFCCurrentStep=> ST03_Ruestsatz[1].SFCCurrentStep,
		SFCTime=>ST03_Ruestsatz[1].SFCTime );
	ST03_72pol_Zufuehrung.FB_CurrentStepHistorie(st_CurrentStep:=ST03_72pol_Zufuehrung.SFCCurrentStep);

	IF	(ModeSelect.Mode=MODE_AUTO_RUN OR 	ModeSelect.Mode=MODE_STEP_RUN)	AND
		NOT gRunEmpty THEN
		ST03_72pol_Zufuehrung.Start:=TRUE;
	ELSE
		ST03_72pol_Zufuehrung.Start:=FALSE;
	END_IF

(*48pol =============================================================================*)
5832:
	ST03_48pol_Zufuehrung(
		SFCCurrentPOU=> ST03_Ruestsatz[1].SFCCurrentPOU,
		SFCCurrentStep=> ST03_Ruestsatz[1].SFCCurrentStep,
		SFCTime=>ST03_Ruestsatz[1].SFCTime );
	ST03_48pol_Zufuehrung.FB_CurrentStepHistorie(st_CurrentStep:=ST03_48pol_Zufuehrung.SFCCurrentStep);

	IF	(ModeSelect.Mode=MODE_AUTO_RUN OR 	ModeSelect.Mode=MODE_STEP_RUN)	AND
		NOT gRunEmpty THEN
		ST03_48pol_Zufuehrung.Start:=TRUE;
	ELSE
		ST03_48pol_Zufuehrung.Start:=FALSE;
	END_IF

(*268pol =============================================================================*)
5841:
	ST03_268pol_Zufuehrung(
		SFCCurrentPOU=> ST03_Ruestsatz[1].SFCCurrentPOU,
		SFCCurrentStep=> ST03_Ruestsatz[1].SFCCurrentStep,
		SFCTime=>ST03_Ruestsatz[1].SFCTime );
	ST03_268pol_Zufuehrung.FB_CurrentStepHistorie(st_CurrentStep:=ST03_268pol_Zufuehrung.SFCCurrentStep);

	IF	(ModeSelect.Mode=MODE_AUTO_RUN OR 	ModeSelect.Mode=MODE_STEP_RUN)	AND
		NOT gRunEmpty THEN
		ST03_268pol_Zufuehrung.Start:=TRUE;
	ELSE
		ST03_268pol_Zufuehrung.Start:=FALSE;
	END_IF

(*102pol neu =============================================================================*)
4993:
	ST03_102pol_neu_Zufuehrung(
		SFCCurrentPOU=> ST03_Ruestsatz[1].SFCCurrentPOU,
		SFCCurrentStep=> ST03_Ruestsatz[1].SFCCurrentStep,
		SFCTime=>ST03_Ruestsatz[1].SFCTime );
	ST03_102pol_neu_Zufuehrung.FB_CurrentStepHistorie(st_CurrentStep:=ST03_102pol_neu_Zufuehrung.SFCCurrentStep);

	IF	(ModeSelect.Mode=MODE_AUTO_RUN OR 	ModeSelect.Mode=MODE_STEP_RUN)	AND
		NOT gRunEmpty THEN
		ST03_102pol_neu_Zufuehrung.Start:=TRUE;
	ELSE
		ST03_102pol_neu_Zufuehrung.Start:=FALSE;
	END_IF


(*268pol RP=============================================================================*)
5842:
	ST03_268_RP_Zufuehrung(
		SFCCurrentPOU=> ST03_Ruestsatz[1].SFCCurrentPOU,
		SFCCurrentStep=> ST03_Ruestsatz[1].SFCCurrentStep,
		SFCTime=>ST03_Ruestsatz[1].SFCTime );
	ST03_268_RP_Zufuehrung.FB_CurrentStepHistorie(st_CurrentStep:=ST03_268_RP_Zufuehrung.SFCCurrentStep);
	ST03_268_RP_Wendeeinheit(
		SFCCurrentPOU=> ST03_Ruestsatz[2].SFCCurrentPOU,
		SFCCurrentStep=> ST03_Ruestsatz[2].SFCCurrentStep,
		SFCTime=>ST03_Ruestsatz[2].SFCTime );
	ST03_268_RP_Wendeeinheit.FB_CurrentStepHistorie(st_CurrentStep:=ST03_268_RP_Wendeeinheit.SFCCurrentStep);
	IF	(ModeSelect.Mode=MODE_AUTO_RUN OR 	ModeSelect.Mode=MODE_STEP_RUN)	AND
		NOT gRunEmpty THEN
		ST03_268_RP_Zufuehrung.Start:=TRUE;
		ST03_268_RP_Wendeeinheit.Start:=TRUE;
	ELSE
		ST03_268_RP_Zufuehrung.Start:=FALSE;
		ST03_268_RP_Wendeeinheit.Start:=FALSE;
	END_IF

(*91pol =============================================================================*)
379:
ST03_91pol_Zufuehrung(
		SFCCurrentPOU=> ST03_Ruestsatz[1].SFCCurrentPOU,
		SFCCurrentStep=> ST03_Ruestsatz[1].SFCCurrentStep,
		SFCTime=>ST03_Ruestsatz[1].SFCTime );
	ST03_91pol_Zufuehrung.FB_CurrentStepHistorie(st_CurrentStep:=ST03_91pol_Zufuehrung.SFCCurrentStep);

	IF	(ModeSelect.Mode=MODE_AUTO_RUN OR 	ModeSelect.Mode=MODE_STEP_RUN)	AND
		NOT gRunEmpty THEN
		ST03_91pol_Zufuehrung.Start:=TRUE;
	ELSE
		ST03_91pol_Zufuehrung.Start:=FALSE;
	END_IF

(*33pol=============================================================================*)
598:
	ST03_33pol_Zufuehrung(
		SFCCurrentPOU=> ST03_Ruestsatz[1].SFCCurrentPOU,
		SFCCurrentStep=> ST03_Ruestsatz[1].SFCCurrentStep,
		SFCTime=>ST03_Ruestsatz[1].SFCTime );
	ST03_33pol_Zufuehrung.FB_CurrentStepHistorie(st_CurrentStep:=ST03_33pol_Zufuehrung.SFCCurrentStep);

	IF	(ModeSelect.Mode=MODE_AUTO_RUN OR 	ModeSelect.Mode=MODE_STEP_RUN)	AND
		NOT gRunEmpty THEN
		ST03_33pol_Zufuehrung.Start:=TRUE;
	ELSE
		ST03_33pol_Zufuehrung.Start:=FALSE;
	END_IF

END_CASE
FOR i:=1 TO 3 BY 1 DO
	ST03_Ruestsatz[i].b_activ:=ST03_Ruestsatz[i].SFCCurrentPOU='-';
END_FOR

(*IFM Kamera=============================================================================*)
IF 	ModeSelect.Mode=MODE_MANUAL THEN
	Visu.ST02_FDB_55X1_7_JOB_BIT1.BitOutToSet:=TD.IFM_CamProgNo.0;
	Visu.ST02_FDB_55X1_7_JOB_BIT2.BitOutToSet:=TD.IFM_CamProgNo.1;

	Visu.ST02_FDB_56X1_7_JOB_BIT1.BitOutToSet:=TD.IFM_CamProgNo.0;
	Visu.ST02_FDB_56X1_7_JOB_BIT2.BitOutToSet:=TD.IFM_CamProgNo.1;
END_IF
END_PROGRAM

(* POU Stations/ST_03_Ruestsaetze/ST_03_PRGs/ST03_ManRobotSwivelUnit, ST *)
PROGRAM ST03_ManRobotSwivelUnit
VAR
 ToggleSwivelOn		: TP;
 ToggleSwivelOff	: TP;
 ToggleBtnOn  		: BOOL;
 ToggleBtnOff  		: BOOL;

END_VAR
ToggleSwivelOn(In:=ToggleBtnOn,Pt:=T#1s);
ToggleSwivelOff(In:=ToggleBtnOff,Pt:=T#1s);

IF 	Robot01.State = STATE_WAIT THEN
 gManSwivelOnRobot01:=ToggleSwivelOn.Q;
 gManSwivelOffRobot01:=ToggleSwivelOff.Q;
END_IF
END_PROGRAM

(* POU Stations/ST_03_Ruestsaetze/ST_03_SFCs/Zufuehrungen/ST03_154pol_Zufuehrung, SFC *)
 PROGRAM ST03_154pol_Zufuehrung
VAR_OUTPUT
	SFCCurrentPOU			: STRING:='ST03_154pol_Zufuehrung';
	SFCCurrentStep			: STRING:='';
	FB_CurrentStepHistorie	: FB_CurrentStepHistorie;
	SFCTime					: DINT;
	State   				: StateObject	:= STATE_WAIT;
	Result  				: StateResult;
END_VAR
VAR_INPUT
	Start					:BOOL;
END_VAR
VAR
	MsgOK				: BOOL;
	MsgCancel			: BOOL;
	SFCRun				: BOOL;
	SFCTimeStart		: TIME;
	Delay				: TON;
	(* Userdefinded area *)

END_VAR
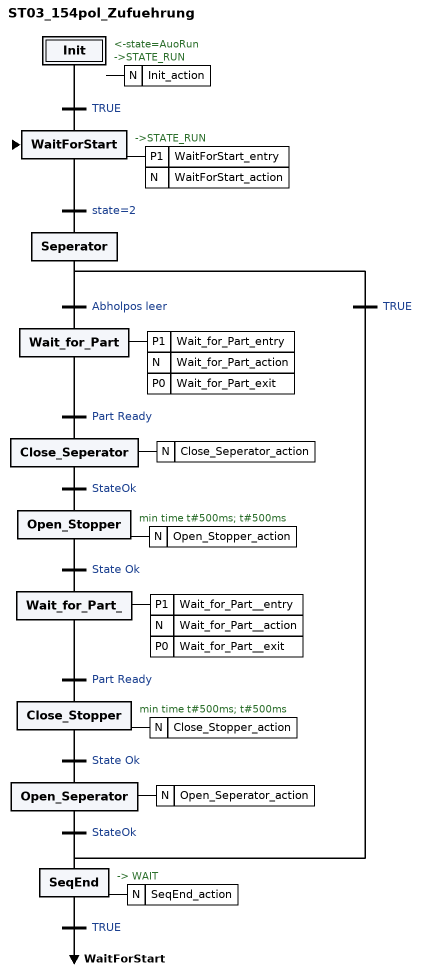
INITIAL_STEP Init: (* <-state=AuoRun / ->STATE_RUN *)
	Init_action(N);
END_STEP
TRANSITION FROM Init TO WaitForStart := TRUE;
END_TRANSITION
STEP WaitForStart: (* ->STATE_RUN *)
	WaitForStart_entry(P1);
	WaitForStart_action(N);
END_STEP
TRANSITION FROM WaitForStart TO Seperator := state=2;
END_TRANSITION
STEP Seperator:
END_STEP
TRANSITION FROM Seperator TO Wait_for_Part := Abholpos leer;
END_TRANSITION
TRANSITION FROM Seperator TO SeqEnd := TRUE;
END_TRANSITION
STEP Wait_for_Part:
	Wait_for_Part_entry(P1);
	Wait_for_Part_action(N);
	Wait_for_Part_exit(P0);
END_STEP
TRANSITION FROM Wait_for_Part TO Close_Seperator := Part Ready;
END_TRANSITION
STEP Close_Seperator:
	Close_Seperator_action(N);
END_STEP
TRANSITION FROM Close_Seperator TO Open_Stopper := StateOk;
END_TRANSITION
STEP Open_Stopper: (* min time t#500ms; t#500ms *)
	Open_Stopper_action(N);
END_STEP
TRANSITION FROM Open_Stopper TO Wait_for_Part_ := State Ok;
END_TRANSITION
STEP Wait_for_Part_:
	Wait_for_Part__entry(P1);
	Wait_for_Part__action(N);
	Wait_for_Part__exit(P0);
END_STEP
TRANSITION FROM Wait_for_Part_ TO Close_Stopper := Part Ready;
END_TRANSITION
STEP Close_Stopper: (* min time t#500ms; t#500ms *)
	Close_Stopper_action(N);
END_STEP
TRANSITION FROM Close_Stopper TO Open_Seperator := State Ok;
END_TRANSITION
STEP Open_Seperator:
	Open_Seperator_action(N);
END_STEP
TRANSITION FROM Open_Seperator TO SeqEnd := StateOk;
END_TRANSITION
STEP SeqEnd: (* -> WAIT *)
	SeqEnd_action(N);
END_STEP
TRANSITION FROM SeqEnd TO WaitForStart := TRUE;
END_TRANSITION

ACTION Init_action:
Start:=FALSE;
State:=STATE_WAIT;
MsgOK:=FALSE;
MsgCancel:=FALSE;
SFCRun:=FALSE;
Result:=RESULT_NON;
END_ACTION

ACTION WaitForStart_entry:
;
END_ACTION

ACTION WaitForStart_action:
IF 	Start   THEN
	State:=STATE_RUN;
	Result:=RESULT_NON;
	SFCTimeStart:=TIME();
	Start:=FALSE;
ELSE
	State:=STATE_WAIT;
	MsgOK:=FALSE;
	MsgCancel:=FALSE;
	SFCRun:=FALSE;
END_IF
END_ACTION

ACTION Wait_for_Part_entry:
ProcessMessage01:='';
Delay.IN:=FALSE;
Delay();
END_ACTION

ACTION Wait_for_Part_action:
ProcessMessage01:='1IM6';(*warte auf Teil in Vereinzelung*)
Delay.IN:=ST03_425_B67_7.BitInToCheck; 		 (* Schnittstelle Iso auf Übergabeposition *)
Delay.PT:=T#500ms;
Delay();
END_ACTION

ACTION Wait_for_Part_exit:
ProcessMessage01:='';
END_ACTION

ACTION Close_Seperator_action:
ST03_426_Y68_5.MoveWork:=TRUE;		(* Förderband  Zuführung Vereinzler AST/GST *)
END_ACTION

ACTION Open_Stopper_action:
ST03_426_Y68_6.MoveWork:=TRUE;		(* Förderband  Züführung Stopper AST/GST *)
END_ACTION

ACTION Wait_for_Part__entry:
ProcessMessage01:='';
Delay.IN:=FALSE;
Delay();
END_ACTION

ACTION Wait_for_Part__action:
ProcessMessage01:='1IM6';(*warte auf Teil in Vereinzelung*)
Delay.IN:=ST03_426_B68_4.BitInToCheck; 		 (* Schnittstelle Iso auf Übergabeposition *)
Delay.PT:=T#500ms;
Delay();
END_ACTION

ACTION Wait_for_Part__exit:
ProcessMessage01:='';
END_ACTION

ACTION Close_Stopper_action:
ST03_426_Y68_6.MoveInit:=TRUE;		(* Förderband  Züführung Stopper AST/GST *)
END_ACTION

ACTION Open_Seperator_action:
ST03_426_Y68_5.MoveInit:=TRUE;		(* Förderband  Zuführung Vereinzler AST/GST *)
END_ACTION

ACTION SeqEnd_action:
SFCTime:=TIME_TO_DINT(TIME()-SFCTimeStart);
State:=STATE_WAIT;
END_ACTION

TRANSITION Abholpos leer:
NOT  ST03_426_B68_4.BitInToCheck
END_TRANSITION

TRANSITION Part Ready:
Delay.Q AND
NOT ST03_426_B68_4.BitInToCheck	AND		(*  Züführung  ISK auf Übergabeposition Roboter Palettierer*)
ST03_425_B67_7.BitInToCheck	AND	(*  ISK anwesend am Vereinzler*)
Robot01.ActualArea <> 4
END_TRANSITION

TRANSITION StateOk:
ST03_426_Y68_5.State=STATE_OK 	(* Förderband  Zuführung Vereinzler AST/GST *)

(*ST03_426_B68_4.BitInToCheck	AND		(*  Züführung  ISK auf Übergabeposition Roboter Palettierer*)
NOT ST03_425_B67_7.BitInToCheck AND	(*  ISK anwesend am Vereinzler*)
gTipImp*)
END_TRANSITION

TRANSITION State Ok:
ST03_426_Y68_6.State=STATE_OK 	(* Förderband  Züführung Stopper AST/GST *)
END_TRANSITION

TRANSITION Part Ready:
Delay.Q AND
(*NOT ST03_426_B68_4.BitInToCheck	AND		(*  Züführung  ISK auf Übergabeposition Roboter Palettierer*)
ST03_425_B67_7.BitInToCheck	AND*)	(*  ISK anwesend am Vereinzler*)
Robot01.ActualArea <> 4
END_TRANSITION

TRANSITION State Ok:
ST03_426_Y68_6.State=STATE_OK 	(* Förderband  Züführung Stopper AST/GST *)
END_TRANSITION

TRANSITION StateOk:
ST03_426_Y68_5.State=STATE_OK 	(* Förderband  Zuführung Vereinzler AST/GST *)

(*ST03_426_B68_4.BitInToCheck	AND		(*  Züführung  ISK auf Übergabeposition Roboter Palettierer*)
NOT ST03_425_B67_7.BitInToCheck AND	(*  ISK anwesend am Vereinzler*)
gTipImp*)
END_TRANSITION
END_PROGRAM

(* POU Stations/ST_03_Ruestsaetze/ST_03_SFCs/Zufuehrungen/ST03_154_RP_Zufuehrung, SFC *)
 PROGRAM ST03_154_RP_Zufuehrung
VAR_OUTPUT
	SFCCurrentPOU			: STRING:='ST03_154_RP_Zufuehrung';
	SFCCurrentStep			: STRING:='';
	FB_CurrentStepHistorie	: FB_CurrentStepHistorie;
	SFCTime					: DINT;
	State   				: StateObject	:= STATE_WAIT;
	Result  				: StateResult;
END_VAR
VAR_INPUT
	Start					:BOOL;
END_VAR
VAR
	MsgOK				: BOOL;
	MsgCancel			: BOOL;
	SFCRun				: BOOL;
	SFCTimeStart		: TIME;
	(* Userdefinded area *)

END_VAR
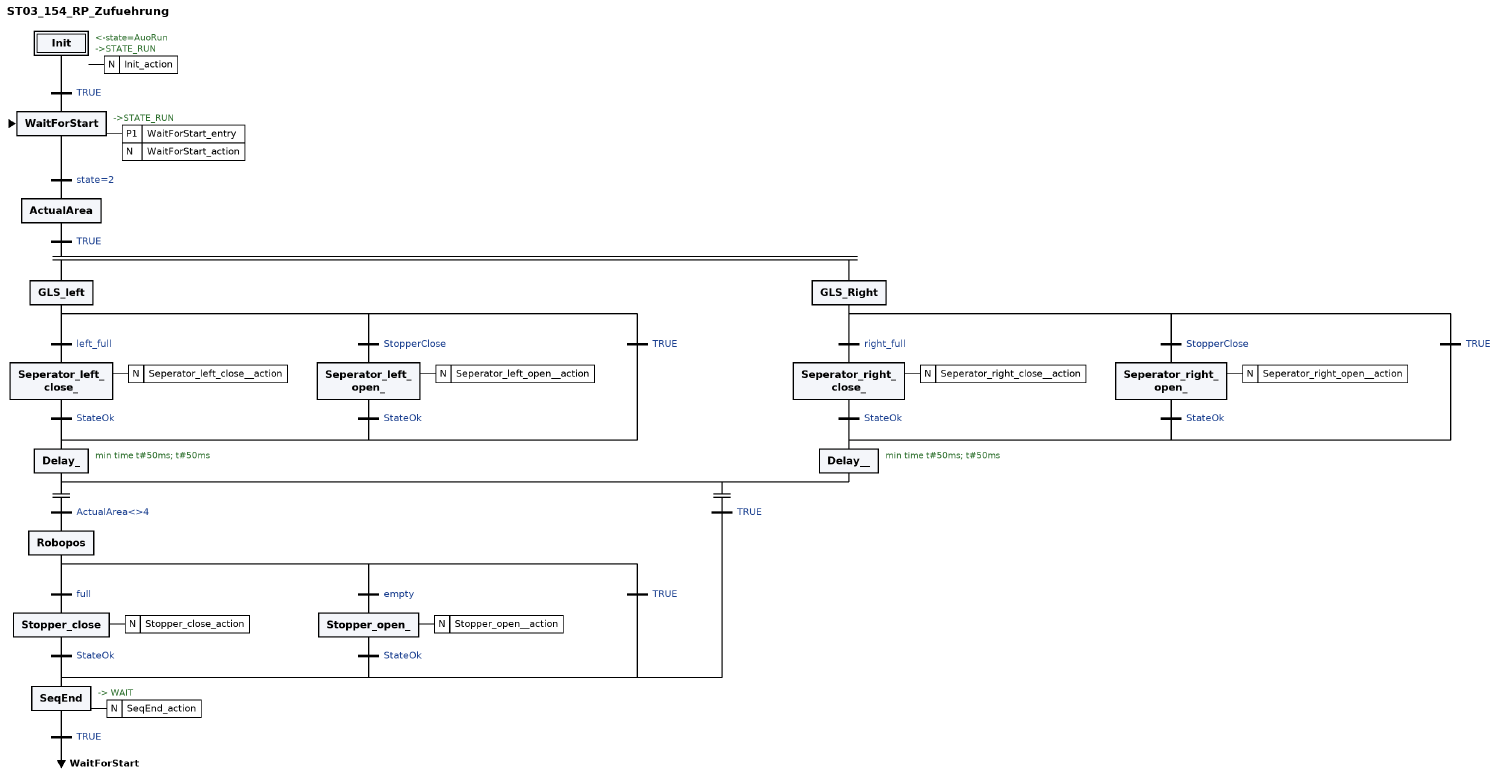
INITIAL_STEP Init: (* <-state=AuoRun / ->STATE_RUN *)
	Init_action(N);
END_STEP
TRANSITION FROM Init TO WaitForStart := TRUE;
END_TRANSITION
STEP WaitForStart: (* ->STATE_RUN *)
	WaitForStart_entry(P1);
	WaitForStart_action(N);
END_STEP
TRANSITION FROM WaitForStart TO ActualArea := state=2;
END_TRANSITION
STEP ActualArea:
END_STEP
TRANSITION FROM ActualArea TO (GLS_left, GLS_Right) := TRUE;
END_TRANSITION
STEP GLS_left:
END_STEP
TRANSITION FROM GLS_left TO Seperator_left_close_ := left_full;
END_TRANSITION
TRANSITION FROM GLS_left TO Seperator_left_open_ := StopperClose;
END_TRANSITION
TRANSITION FROM GLS_left TO Delay_ := TRUE;
END_TRANSITION
STEP Seperator_left_close_:
	Seperator_left_close__action(N);
END_STEP
TRANSITION FROM Seperator_left_close_ TO Delay_ := StateOk;
END_TRANSITION
STEP Seperator_left_open_:
	Seperator_left_open__action(N);
END_STEP
TRANSITION FROM Seperator_left_open_ TO Delay_ := StateOk;
END_TRANSITION
STEP Delay_: (* min time t#50ms; t#50ms *)
END_STEP
STEP GLS_Right:
END_STEP
TRANSITION FROM GLS_Right TO Seperator_right_close_ := right_full;
END_TRANSITION
TRANSITION FROM GLS_Right TO Seperator_right_open_ := StopperClose;
END_TRANSITION
TRANSITION FROM GLS_Right TO Delay__ := TRUE;
END_TRANSITION
STEP Seperator_right_close_:
	Seperator_right_close__action(N);
END_STEP
TRANSITION FROM Seperator_right_close_ TO Delay__ := StateOk;
END_TRANSITION
STEP Seperator_right_open_:
	Seperator_right_open__action(N);
END_STEP
TRANSITION FROM Seperator_right_open_ TO Delay__ := StateOk;
END_TRANSITION
STEP Delay__: (* min time t#50ms; t#50ms *)
END_STEP
TRANSITION FROM (Delay_, Delay__) TO Robopos := ActualArea<>4;
END_TRANSITION
TRANSITION FROM (Delay_, Delay__) TO SeqEnd := TRUE;
END_TRANSITION
STEP Robopos:
END_STEP
TRANSITION FROM Robopos TO Stopper_close := full;
END_TRANSITION
TRANSITION FROM Robopos TO Stopper_open_ := empty;
END_TRANSITION
TRANSITION FROM Robopos TO SeqEnd := TRUE;
END_TRANSITION
STEP Stopper_close:
	Stopper_close_action(N);
END_STEP
TRANSITION FROM Stopper_close TO SeqEnd := StateOk;
END_TRANSITION
STEP Stopper_open_:
	Stopper_open__action(N);
END_STEP
TRANSITION FROM Stopper_open_ TO SeqEnd := StateOk;
END_TRANSITION
STEP SeqEnd: (* -> WAIT *)
	SeqEnd_action(N);
END_STEP
TRANSITION FROM SeqEnd TO WaitForStart := TRUE;
END_TRANSITION

ACTION Init_action:
Start:=FALSE;
State:=STATE_WAIT;
MsgOK:=FALSE;
MsgCancel:=FALSE;
SFCRun:=FALSE;
Result:=RESULT_NON;
END_ACTION

ACTION WaitForStart_entry:
;
END_ACTION

ACTION WaitForStart_action:
IF 	Start   THEN
	State:=STATE_RUN;
	Result:=RESULT_NON;
	SFCTimeStart:=TIME();
	Start:=FALSE;
ELSE
	State:=STATE_WAIT;
	MsgOK:=FALSE;
	MsgCancel:=FALSE;
	SFCRun:=FALSE;
END_IF
END_ACTION

ACTION Seperator_left_close__action:
ST03_419_Y61_5.MoveWork:=TRUE;	(* Förderband linke Zuführung Vereinzler AST/GST *)
END_ACTION

ACTION Seperator_left_open__action:
ST03_419_Y61_5.MoveInit:=TRUE;		(* Förderband linke Zuführung Vereinzler AST/GST *)
END_ACTION

ACTION Seperator_right_close__action:
ST03_419_Y61_6.MoveWork:=TRUE;	(* Förderband rechts Zuführung Vereinzler AST/GST *)
END_ACTION

ACTION Seperator_right_open__action:
ST03_419_Y61_6.MoveInit:=TRUE;			(* Förderband rechts Zuführung Vereinzler AST/GST *)
END_ACTION

ACTION Stopper_close_action:
ST03_419_Y61_7.MoveInit:=TRUE;		(* Förderband links/rechts Züführung Stopper AST/GST *)
END_ACTION

ACTION Stopper_open__action:
ST03_419_Y61_7.MoveWork:=TRUE;		(* Förderband links/rechts Züführung Stopper AST/GST *)
END_ACTION

ACTION SeqEnd_action:
SFCTime:=TIME_TO_DINT(TIME()-SFCTimeStart);
State:=STATE_WAIT;
END_ACTION

TRANSITION left_full:
ST03_419_B61_0.BitInToCheck			(*  Förderband Zuführung links ISK anwesend zum Vereinzeln*)
END_TRANSITION

TRANSITION StateOk:
ST03_419_Y61_5.State=STATE_OK
AND
gTipImp
END_TRANSITION

TRANSITION StopperClose:
NOT ST03_418_B60_4.ValveSensor AND
ST03_418_B60_5.ValveSensor
END_TRANSITION

TRANSITION StateOk:
ST03_419_Y61_5.State=STATE_OK 	(* Förderband  Zuführung Vereinzler AST/GST *)
AND
gTipImp
END_TRANSITION

TRANSITION right_full:
ST03_419_B61_1.BitInToCheck			(*  Förderband Zuführung rechts ISK anwesend zum Vereinzeln*)
END_TRANSITION

TRANSITION StateOk:
ST03_419_Y61_6.State=STATE_OK (* Förderband rechts Zuführung Vereinzler AST/GST *)
AND
gTipImp
END_TRANSITION

TRANSITION StopperClose:
NOT ST03_418_B60_4.ValveSensor AND
ST03_418_B60_5.ValveSensor
END_TRANSITION

TRANSITION StateOk:
ST03_419_Y61_6.State=STATE_OK 	(* Förderband rechts Zuführung Vereinzler AST/GST *)
AND
gTipImp
END_TRANSITION

TRANSITION ActualArea<>4:
Robot01.ActualArea <> 4
END_TRANSITION

TRANSITION full:
ST03_419_B61_2.BitInToCheck AND 	(*  Züführung links ISK auf Übergabeposition Roboter Palettierer*)
ST03_419_B61_3.BitInToCheck		(*  Züführung rechts ISK auf Übergabeposition Roboter Palettierer*)
END_TRANSITION

TRANSITION StateOk:
ST03_419_Y61_7.State=STATE_OK 	(* Förderband  Zuführung Vereinzler AST/GST *)
AND
gTipImp
END_TRANSITION

TRANSITION empty:
NOT ST03_419_B61_2.BitInToCheck AND 	(*  Züführung links ISK auf Übergabeposition Roboter Palettierer*)
NOT ST03_419_B61_3.BitInToCheck		(*  Züführung rechts ISK auf Übergabeposition Roboter Palettierer*)
END_TRANSITION

TRANSITION StateOk:
ST03_419_Y61_7.State=STATE_OK 	(* Förderband  Zuführung Vereinzler AST/GST *)
AND
gTipImp
END_TRANSITION
END_PROGRAM

(* POU Stations/ST_03_Ruestsaetze/ST_03_SFCs/Zufuehrungen/ST03_206pol_Zufuehrung, SFC *)
 PROGRAM ST03_206pol_Zufuehrung
VAR_OUTPUT
	SFCCurrentPOU			: STRING:='ST03_206pol_Zufuehrung';
	SFCCurrentStep			: STRING:='';
	FB_CurrentStepHistorie	: FB_CurrentStepHistorie;
	SFCTime					: DINT;
	State   				: StateObject	:= STATE_WAIT;
	Result  				: StateResult;
END_VAR
VAR_INPUT
	Start					:BOOL;
END_VAR
VAR
	MsgOK				: BOOL;
	MsgCancel			: BOOL;
	SFCRun				: BOOL;
	SFCTimeStart		: TIME;
	Delay				: TON;
	(* Userdefinded area *)

END_VAR
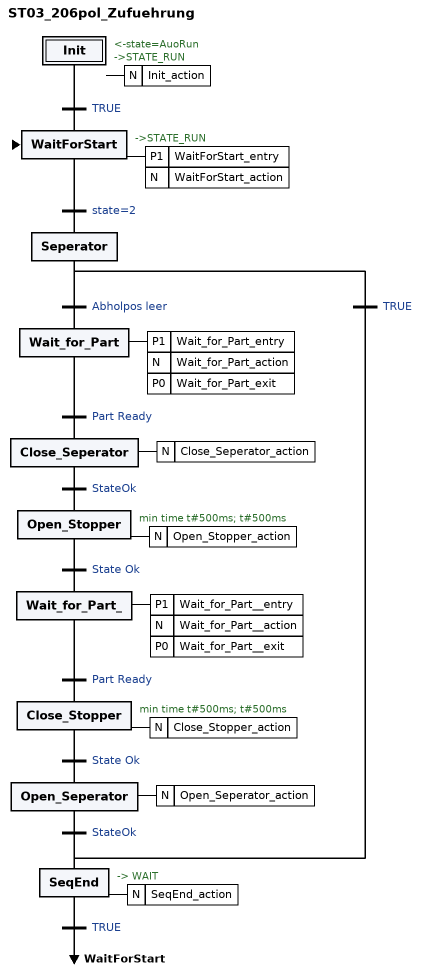
INITIAL_STEP Init: (* <-state=AuoRun / ->STATE_RUN *)
	Init_action(N);
END_STEP
TRANSITION FROM Init TO WaitForStart := TRUE;
END_TRANSITION
STEP WaitForStart: (* ->STATE_RUN *)
	WaitForStart_entry(P1);
	WaitForStart_action(N);
END_STEP
TRANSITION FROM WaitForStart TO Seperator := state=2;
END_TRANSITION
STEP Seperator:
END_STEP
TRANSITION FROM Seperator TO Wait_for_Part := Abholpos leer;
END_TRANSITION
TRANSITION FROM Seperator TO SeqEnd := TRUE;
END_TRANSITION
STEP Wait_for_Part:
	Wait_for_Part_entry(P1);
	Wait_for_Part_action(N);
	Wait_for_Part_exit(P0);
END_STEP
TRANSITION FROM Wait_for_Part TO Close_Seperator := Part Ready;
END_TRANSITION
STEP Close_Seperator:
	Close_Seperator_action(N);
END_STEP
TRANSITION FROM Close_Seperator TO Open_Stopper := StateOk;
END_TRANSITION
STEP Open_Stopper: (* min time t#500ms; t#500ms *)
	Open_Stopper_action(N);
END_STEP
TRANSITION FROM Open_Stopper TO Wait_for_Part_ := State Ok;
END_TRANSITION
STEP Wait_for_Part_:
	Wait_for_Part__entry(P1);
	Wait_for_Part__action(N);
	Wait_for_Part__exit(P0);
END_STEP
TRANSITION FROM Wait_for_Part_ TO Close_Stopper := Part Ready;
END_TRANSITION
STEP Close_Stopper: (* min time t#500ms; t#500ms *)
	Close_Stopper_action(N);
END_STEP
TRANSITION FROM Close_Stopper TO Open_Seperator := State Ok;
END_TRANSITION
STEP Open_Seperator:
	Open_Seperator_action(N);
END_STEP
TRANSITION FROM Open_Seperator TO SeqEnd := StateOk;
END_TRANSITION
STEP SeqEnd: (* -> WAIT *)
	SeqEnd_action(N);
END_STEP
TRANSITION FROM SeqEnd TO WaitForStart := TRUE;
END_TRANSITION

ACTION Init_action:
Start:=FALSE;
State:=STATE_WAIT;
MsgOK:=FALSE;
MsgCancel:=FALSE;
SFCRun:=FALSE;
Result:=RESULT_NON;
END_ACTION

ACTION WaitForStart_entry:
;
END_ACTION

ACTION WaitForStart_action:
IF 	Start   THEN
	State:=STATE_RUN;
	Result:=RESULT_NON;
	SFCTimeStart:=TIME();
	Start:=FALSE;
ELSE
	State:=STATE_WAIT;
	MsgOK:=FALSE;
	MsgCancel:=FALSE;
	SFCRun:=FALSE;
END_IF
END_ACTION

ACTION Wait_for_Part_entry:
ProcessMessage01:='';
Delay.IN:=FALSE;
Delay();
END_ACTION

ACTION Wait_for_Part_action:
ProcessMessage01:='1IM6';(*warte auf Teil in Vereinzelung*)
Delay.IN:=ST03_435_B67_7.BitInToCheck; 		 (* Schnittstelle Iso auf Übergabeposition *)
Delay.PT:=T#500ms;
Delay();
END_ACTION

ACTION Wait_for_Part_exit:
ProcessMessage01:='';
END_ACTION

ACTION Close_Seperator_action:
ST03_437_Y68_5.MoveWork:=TRUE;		(* Förderband  Zuführung Vereinzler AST/GST *)
END_ACTION

ACTION Open_Stopper_action:
ST03_437_Y68_6.MoveWork:=TRUE;		(* Förderband  Züführung Stopper AST/GST *)
END_ACTION

ACTION Wait_for_Part__entry:
ProcessMessage01:='';
Delay.IN:=FALSE;
Delay();
END_ACTION

ACTION Wait_for_Part__action:
ProcessMessage01:='1IM6';(*warte auf Teil in Vereinzelung*)
Delay.IN:=	ST03_Init_AbholPos.RoboPos31 OR
			ST03_Init_AbholPos.RoboPos35 OR
			NOT ST03_437_B68_4.BitInToCheck;
Delay.PT:=T#500ms;
Delay();
END_ACTION

ACTION Wait_for_Part__exit:
ProcessMessage01:='';
END_ACTION

ACTION Close_Stopper_action:
ST03_437_Y68_6.MoveInit:=TRUE;		(* Förderband  Züführung Stopper AST/GST *)
END_ACTION

ACTION Open_Seperator_action:
ST03_437_Y68_5.MoveInit:=TRUE;		(* Förderband  Zuführung Vereinzler AST/GST *)
END_ACTION

ACTION SeqEnd_action:
SFCTime:=TIME_TO_DINT(TIME()-SFCTimeStart);
State:=STATE_WAIT;
END_ACTION

TRANSITION Abholpos leer:
NOT ST03_Init_AbholPos.RoboPos31 AND
NOT ST03_Init_AbholPos.RoboPos35
END_TRANSITION

TRANSITION Part Ready:
Delay.Q AND
ST03_435_B67_7.BitInToCheck	AND	(*  ISK anwesend am Stoper*)
Robot01.ActualArea <> 4
END_TRANSITION

TRANSITION StateOk:
ST03_437_Y68_5.State=STATE_OK 	(* Förderband  Zuführung Vereinzler AST/GST *)

(*ST03_426_B68_4.BitInToCheck	AND		(*  Züführung  ISK auf Übergabeposition Roboter Palettierer*)
NOT ST03_425_B67_7.BitInToCheck AND	(*  ISK anwesend am Vereinzler*)
gTipImp*)
END_TRANSITION

TRANSITION State Ok:
ST03_437_Y68_6.State=STATE_OK 	(* Förderband  Züführung Stopper AST/GST *)
END_TRANSITION

TRANSITION Part Ready:
Delay.Q AND
(ST03_Init_AbholPos.RoboPos31 OR
ST03_Init_AbholPos.RoboPos35) AND
Robot01.ActualArea <> 4
END_TRANSITION

TRANSITION State Ok:
ST03_437_Y68_6.State=STATE_OK 	(* Förderband  Züführung Stopper AST/GST *)
END_TRANSITION

TRANSITION StateOk:
ST03_437_Y68_5.State=STATE_OK 	(* Förderband  Zuführung Vereinzler AST/GST *)
END_TRANSITION
END_PROGRAM

(* POU Stations/ST_03_Ruestsaetze/ST_03_SFCs/Zufuehrungen/ST03_92pol_Zufuehrung, SFC *)
 PROGRAM ST03_92pol_Zufuehrung
VAR_OUTPUT
	SFCCurrentPOU			: STRING:='ST03_92pol_Zufuehrung';
	SFCCurrentStep			: STRING:='';
	FB_CurrentStepHistorie	: FB_CurrentStepHistorie;
	SFCTime					: DINT;
	State   				: StateObject	:= STATE_WAIT;
	Result  				: StateResult;
END_VAR
VAR_INPUT
	Start					:BOOL;
END_VAR
VAR
	MsgOK				: BOOL;
	MsgCancel			: BOOL;
	SFCRun				: BOOL;
	SFCTimeStart		: TIME;
	Delay				: TON;
	(* Userdefinded area *)

END_VAR
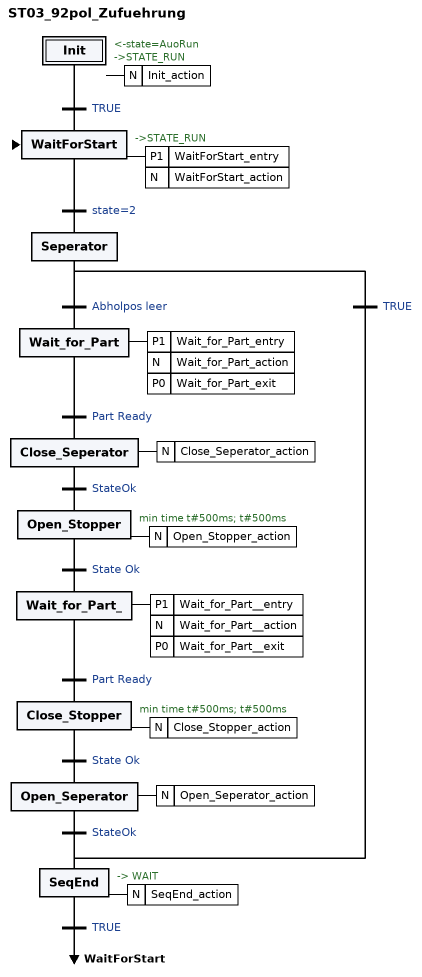
INITIAL_STEP Init: (* <-state=AuoRun / ->STATE_RUN *)
	Init_action(N);
END_STEP
TRANSITION FROM Init TO WaitForStart := TRUE;
END_TRANSITION
STEP WaitForStart: (* ->STATE_RUN *)
	WaitForStart_entry(P1);
	WaitForStart_action(N);
END_STEP
TRANSITION FROM WaitForStart TO Seperator := state=2;
END_TRANSITION
STEP Seperator:
END_STEP
TRANSITION FROM Seperator TO Wait_for_Part := Abholpos leer;
END_TRANSITION
TRANSITION FROM Seperator TO SeqEnd := TRUE;
END_TRANSITION
STEP Wait_for_Part:
	Wait_for_Part_entry(P1);
	Wait_for_Part_action(N);
	Wait_for_Part_exit(P0);
END_STEP
TRANSITION FROM Wait_for_Part TO Close_Seperator := Part Ready;
END_TRANSITION
STEP Close_Seperator:
	Close_Seperator_action(N);
END_STEP
TRANSITION FROM Close_Seperator TO Open_Stopper := StateOk;
END_TRANSITION
STEP Open_Stopper: (* min time t#500ms; t#500ms *)
	Open_Stopper_action(N);
END_STEP
TRANSITION FROM Open_Stopper TO Wait_for_Part_ := State Ok;
END_TRANSITION
STEP Wait_for_Part_:
	Wait_for_Part__entry(P1);
	Wait_for_Part__action(N);
	Wait_for_Part__exit(P0);
END_STEP
TRANSITION FROM Wait_for_Part_ TO Close_Stopper := Part Ready;
END_TRANSITION
STEP Close_Stopper: (* min time t#500ms; t#500ms *)
	Close_Stopper_action(N);
END_STEP
TRANSITION FROM Close_Stopper TO Open_Seperator := State Ok;
END_TRANSITION
STEP Open_Seperator:
	Open_Seperator_action(N);
END_STEP
TRANSITION FROM Open_Seperator TO SeqEnd := StateOk;
END_TRANSITION
STEP SeqEnd: (* -> WAIT *)
	SeqEnd_action(N);
END_STEP
TRANSITION FROM SeqEnd TO WaitForStart := TRUE;
END_TRANSITION

ACTION Init_action:
Start:=FALSE;
State:=STATE_WAIT;
MsgOK:=FALSE;
MsgCancel:=FALSE;
SFCRun:=FALSE;
Result:=RESULT_NON;
END_ACTION

ACTION WaitForStart_entry:
;
END_ACTION

ACTION WaitForStart_action:
IF 	Start   THEN
	State:=STATE_RUN;
	Result:=RESULT_NON;
	SFCTimeStart:=TIME();
	Start:=FALSE;
ELSE
	State:=STATE_WAIT;
	MsgOK:=FALSE;
	MsgCancel:=FALSE;
	SFCRun:=FALSE;
END_IF
END_ACTION

ACTION Wait_for_Part_entry:
ProcessMessage01:='';
Delay.IN:=FALSE;
Delay();
END_ACTION

ACTION Wait_for_Part_action:
ProcessMessage01:='1IM6';(*warte auf Teil in Vereinzelung*)
Delay.IN:=ST03_444_B69_7.BitInToCheck; 		 (* Schnittstelle Iso auf Übergabeposition *)
Delay.PT:=T#500ms;
Delay();
END_ACTION

ACTION Wait_for_Part_exit:
ProcessMessage01:='';
END_ACTION

ACTION Close_Seperator_action:
ST03_446_Y70_5.MoveWork:=TRUE;		(* Förderband  Zuführung Vereinzler AST/GST *)
END_ACTION

ACTION Open_Stopper_action:
ST03_446_Y70_6.MoveWork:=TRUE;		(* Förderband  Züführung Stopper AST/GST *)
END_ACTION

ACTION Wait_for_Part__entry:
ProcessMessage01:='';
Delay.IN:=FALSE;
Delay();
END_ACTION

ACTION Wait_for_Part__action:
ProcessMessage01:='1IM6';(*warte auf Teil in Vereinzelung*)
Delay.IN:=ST03_446_B70_4.BitInToCheck; 		 (* Schnittstelle Iso auf Übergabeposition Roboter *)
Delay.PT:=T#500ms;
Delay();
END_ACTION

ACTION Wait_for_Part__exit:
ProcessMessage01:='';
END_ACTION

ACTION Close_Stopper_action:
ST03_446_Y70_6.MoveInit:=TRUE;		(* Förderband  Züführung Stopper AST/GST *)
END_ACTION

ACTION Open_Seperator_action:
ST03_446_Y70_5.MoveInit:=TRUE;		(* Förderband  Zuführung Vereinzler AST/GST *)
END_ACTION

ACTION SeqEnd_action:
SFCTime:=TIME_TO_DINT(TIME()-SFCTimeStart);
State:=STATE_WAIT;
END_ACTION

TRANSITION Abholpos leer:
NOT  ST03_446_B70_4.BitInToCheck
END_TRANSITION

TRANSITION Part Ready:
Delay.Q AND
NOT ST03_446_B70_4.BitInToCheck	AND		(*  Züführung  ISK auf Übergabeposition Roboter Palettierer*)
ST03_444_B69_7.BitInToCheck	AND	(*  ISK anwesend am Vereinzler*)
Robot01.ActualArea <> 4
END_TRANSITION

TRANSITION StateOk:
ST03_446_Y70_5.State=STATE_OK 	(* Förderband  Zuführung Vereinzler AST/GST *)

(*ST03_426_B68_4.BitInToCheck	AND		(*  Züführung  ISK auf Übergabeposition Roboter Palettierer*)
NOT ST03_425_B67_7.BitInToCheck AND	(*  ISK anwesend am Vereinzler*)
gTipImp*)
END_TRANSITION

TRANSITION State Ok:
ST03_446_Y70_6.State=STATE_OK 	(* Förderband  Züführung Stopper AST/GST *)
END_TRANSITION

TRANSITION Part Ready:
Delay.Q AND
(*NOT ST03_426_B68_4.BitInToCheck	AND		(*  Züführung  ISK auf Übergabeposition Roboter Palettierer*)
ST03_425_B67_7.BitInToCheck	AND*)	(*  ISK anwesend am Vereinzler*)
Robot01.ActualArea <> 4
END_TRANSITION

TRANSITION State Ok:
ST03_446_Y70_6.State=STATE_OK 	(* Förderband  Züführung Stopper AST/GST *)
END_TRANSITION

TRANSITION StateOk:
ST03_446_Y70_5.State=STATE_OK 	(* Förderband  Zuführung Vereinzler AST/GST *)

(*ST03_426_B68_4.BitInToCheck	AND		(*  Züführung  ISK auf Übergabeposition Roboter Palettierer*)
NOT ST03_425_B67_7.BitInToCheck AND	(*  ISK anwesend am Vereinzler*)
gTipImp*)
END_TRANSITION
END_PROGRAM

(* POU Stations/ST_03_Ruestsaetze/ST_03_SFCs/Zufuehrungen/ST03_124pol_Zufuehrung, SFC *)
 PROGRAM ST03_124pol_Zufuehrung
VAR_OUTPUT
	SFCCurrentPOU			: STRING:='ST03_124pol_Zufuehrung';
	SFCCurrentStep			: STRING:='';
	FB_CurrentStepHistorie	: FB_CurrentStepHistorie;
	SFCTime					: DINT;
	State   				: StateObject	:= STATE_WAIT;
	Result  				: StateResult;
END_VAR
VAR_INPUT
	Start					:BOOL;
END_VAR
VAR
	MsgOK				: BOOL;
	MsgCancel			: BOOL;
	SFCRun				: BOOL;
	SFCTimeStart		: TIME;
	Delay				: TON;
	(* Userdefinded area *)

END_VAR
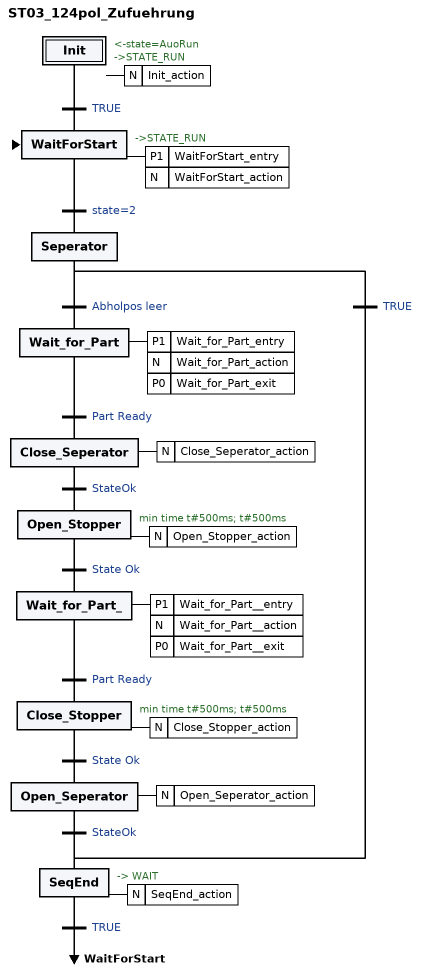
INITIAL_STEP Init: (* <-state=AuoRun / ->STATE_RUN *)
	Init_action(N);
END_STEP
TRANSITION FROM Init TO WaitForStart := TRUE;
END_TRANSITION
STEP WaitForStart: (* ->STATE_RUN *)
	WaitForStart_entry(P1);
	WaitForStart_action(N);
END_STEP
TRANSITION FROM WaitForStart TO Seperator := state=2;
END_TRANSITION
STEP Seperator:
END_STEP
TRANSITION FROM Seperator TO Wait_for_Part := Abholpos leer;
END_TRANSITION
TRANSITION FROM Seperator TO SeqEnd := TRUE;
END_TRANSITION
STEP Wait_for_Part:
	Wait_for_Part_entry(P1);
	Wait_for_Part_action(N);
	Wait_for_Part_exit(P0);
END_STEP
TRANSITION FROM Wait_for_Part TO Close_Seperator := Part Ready;
END_TRANSITION
STEP Close_Seperator:
	Close_Seperator_action(N);
END_STEP
TRANSITION FROM Close_Seperator TO Open_Stopper := StateOk;
END_TRANSITION
STEP Open_Stopper: (* min time t#500ms; t#500ms *)
	Open_Stopper_action(N);
END_STEP
TRANSITION FROM Open_Stopper TO Wait_for_Part_ := State Ok;
END_TRANSITION
STEP Wait_for_Part_:
	Wait_for_Part__entry(P1);
	Wait_for_Part__action(N);
	Wait_for_Part__exit(P0);
END_STEP
TRANSITION FROM Wait_for_Part_ TO Close_Stopper := Part Ready;
END_TRANSITION
STEP Close_Stopper: (* min time t#500ms; t#500ms *)
	Close_Stopper_action(N);
END_STEP
TRANSITION FROM Close_Stopper TO Open_Seperator := State Ok;
END_TRANSITION
STEP Open_Seperator:
	Open_Seperator_action(N);
END_STEP
TRANSITION FROM Open_Seperator TO SeqEnd := StateOk;
END_TRANSITION
STEP SeqEnd: (* -> WAIT *)
	SeqEnd_action(N);
END_STEP
TRANSITION FROM SeqEnd TO WaitForStart := TRUE;
END_TRANSITION

ACTION Init_action:
Start:=FALSE;
State:=STATE_WAIT;
MsgOK:=FALSE;
MsgCancel:=FALSE;
SFCRun:=FALSE;
Result:=RESULT_NON;
END_ACTION

ACTION WaitForStart_entry:
;
END_ACTION

ACTION WaitForStart_action:
IF 	Start   THEN
	State:=STATE_RUN;
	Result:=RESULT_NON;
	SFCTimeStart:=TIME();
	Start:=FALSE;
ELSE
	State:=STATE_WAIT;
	MsgOK:=FALSE;
	MsgCancel:=FALSE;
	SFCRun:=FALSE;
END_IF
END_ACTION

ACTION Wait_for_Part_entry:
ProcessMessage01:='';
Delay.IN:=FALSE;
Delay();
END_ACTION

ACTION Wait_for_Part_action:
ProcessMessage01:='1IM6';(*warte auf Teil in Vereinzelung*)
Delay.IN:=ST03_451_B69_7.BitInToCheck; 		 (* Schnittstelle Iso auf Übergabeposition *)
Delay.PT:=T#500ms;
Delay();
END_ACTION

ACTION Wait_for_Part_exit:
ProcessMessage01:='';
END_ACTION

ACTION Close_Seperator_action:
ST03_453_Y70_5.MoveWork:=TRUE;		(* Förderband  Zuführung Vereinzler AST/GST *)
END_ACTION

ACTION Open_Stopper_action:
ST03_453_Y70_6.MoveWork:=TRUE;		(* Förderband  Züführung Stopper AST/GST *)
END_ACTION

ACTION Wait_for_Part__entry:
ProcessMessage01:='';
Delay.IN:=FALSE;
Delay();
END_ACTION

ACTION Wait_for_Part__action:
ProcessMessage01:='1IM6';(*warte auf Teil in Vereinzelung*)
Delay.IN:=ST03_453_B70_4.BitInToCheck; 		 (* Schnittstelle Iso auf Übergabeposition Roboter *)
Delay.PT:=T#500ms;
Delay();
END_ACTION

ACTION Wait_for_Part__exit:
ProcessMessage01:='';
END_ACTION

ACTION Close_Stopper_action:
ST03_453_Y70_6.MoveInit:=TRUE;		(* Förderband  Züführung Stopper AST/GST *)
END_ACTION

ACTION Open_Seperator_action:
ST03_453_Y70_5.MoveInit:=TRUE;		(* Förderband  Zuführung Vereinzler AST/GST *)
END_ACTION

ACTION SeqEnd_action:
SFCTime:=TIME_TO_DINT(TIME()-SFCTimeStart);
State:=STATE_WAIT;
END_ACTION

TRANSITION Abholpos leer:
NOT  ST03_453_B70_4.BitInToCheck
END_TRANSITION

TRANSITION Part Ready:
Delay.Q AND
NOT ST03_453_B70_4.BitInToCheck	AND		(*  Züführung  ISK auf Übergabeposition Roboter Palettierer*)
ST03_451_B69_7.BitInToCheck	AND	(*  ISK anwesend am Vereinzler*)
Robot01.ActualArea <> 4
END_TRANSITION

TRANSITION StateOk:
ST03_453_Y70_5.State=STATE_OK 	(* Förderband  Zuführung Vereinzler AST/GST *)

(*ST03_426_B68_4.BitInToCheck	AND		(*  Züführung  ISK auf Übergabeposition Roboter Palettierer*)
NOT ST03_425_B67_7.BitInToCheck AND	(*  ISK anwesend am Vereinzler*)
gTipImp*)
END_TRANSITION

TRANSITION State Ok:
ST03_453_Y70_6.State=STATE_OK 	(* Förderband  Züführung Stopper AST/GST *)
END_TRANSITION

TRANSITION Part Ready:
Delay.Q AND
(*NOT ST03_426_B68_4.BitInToCheck	AND		(*  Züführung  ISK auf Übergabeposition Roboter Palettierer*)
ST03_425_B67_7.BitInToCheck	AND*)	(*  ISK anwesend am Vereinzler*)
Robot01.ActualArea <> 4
END_TRANSITION

TRANSITION State Ok:
ST03_453_Y70_6.State=STATE_OK 	(* Förderband  Züführung Stopper AST/GST *)
END_TRANSITION

TRANSITION StateOk:
ST03_453_Y70_5.State=STATE_OK 	(* Förderband  Zuführung Vereinzler AST/GST *)

(*ST03_426_B68_4.BitInToCheck	AND		(*  Züführung  ISK auf Übergabeposition Roboter Palettierer*)
NOT ST03_425_B67_7.BitInToCheck AND	(*  ISK anwesend am Vereinzler*)
gTipImp*)
END_TRANSITION
END_PROGRAM

(* POU Stations/ST_03_Ruestsaetze/ST_03_SFCs/Zufuehrungen/ST03_46pol_Zufuehrung, SFC *)
 PROGRAM ST03_46pol_Zufuehrung
VAR_OUTPUT
	SFCCurrentPOU			: STRING:='ST03_46pol_Zufuehrung';
	SFCCurrentStep			: STRING:='';
	FB_CurrentStepHistorie	: FB_CurrentStepHistorie;
	SFCTime					: DINT;
	State   				: StateObject	:= STATE_WAIT;
	Result  				: StateResult;
END_VAR
VAR_INPUT
	Start					:BOOL;
END_VAR
VAR
	MsgOK				: BOOL;
	MsgCancel			: BOOL;
	SFCRun				: BOOL;
	SFCTimeStart		: TIME;
	Delay				: TON;
	(* Userdefinded area *)

END_VAR
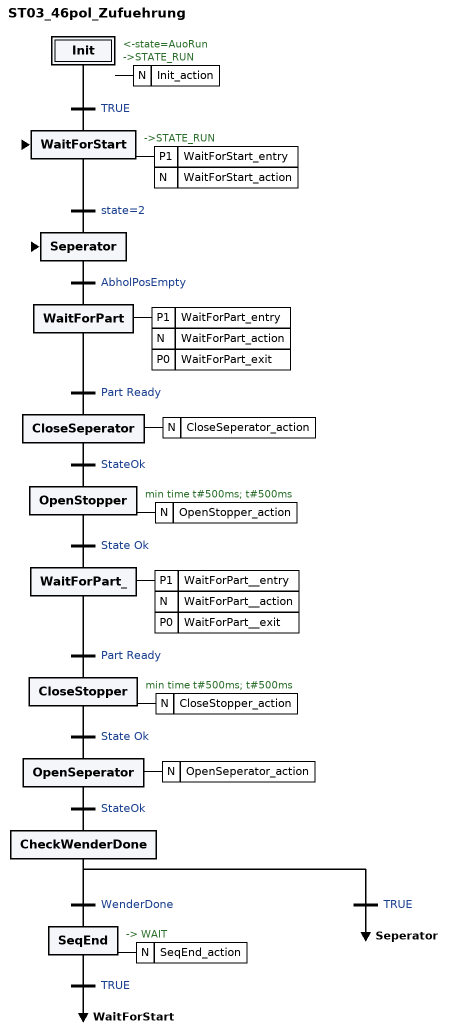
INITIAL_STEP Init: (* <-state=AuoRun / ->STATE_RUN *)
	Init_action(N);
END_STEP
TRANSITION FROM Init TO WaitForStart := TRUE;
END_TRANSITION
STEP WaitForStart: (* ->STATE_RUN *)
	WaitForStart_entry(P1);
	WaitForStart_action(N);
END_STEP
TRANSITION FROM WaitForStart TO Seperator := state=2;
END_TRANSITION
STEP Seperator:
END_STEP
TRANSITION FROM Seperator TO WaitForPart := AbholPosEmpty;
END_TRANSITION
STEP WaitForPart:
	WaitForPart_entry(P1);
	WaitForPart_action(N);
	WaitForPart_exit(P0);
END_STEP
TRANSITION FROM WaitForPart TO CloseSeperator := Part Ready;
END_TRANSITION
STEP CloseSeperator:
	CloseSeperator_action(N);
END_STEP
TRANSITION FROM CloseSeperator TO OpenStopper := StateOk;
END_TRANSITION
STEP OpenStopper: (* min time t#500ms; t#500ms *)
	OpenStopper_action(N);
END_STEP
TRANSITION FROM OpenStopper TO WaitForPart_ := State Ok;
END_TRANSITION
STEP WaitForPart_:
	WaitForPart__entry(P1);
	WaitForPart__action(N);
	WaitForPart__exit(P0);
END_STEP
TRANSITION FROM WaitForPart_ TO CloseStopper := Part Ready;
END_TRANSITION
STEP CloseStopper: (* min time t#500ms; t#500ms *)
	CloseStopper_action(N);
END_STEP
TRANSITION FROM CloseStopper TO OpenSeperator := State Ok;
END_TRANSITION
STEP OpenSeperator:
	OpenSeperator_action(N);
END_STEP
TRANSITION FROM OpenSeperator TO CheckWenderDone := StateOk;
END_TRANSITION
STEP CheckWenderDone:
END_STEP
TRANSITION FROM CheckWenderDone TO SeqEnd := WenderDone;
END_TRANSITION
TRANSITION FROM CheckWenderDone TO Seperator := TRUE;
END_TRANSITION
STEP SeqEnd: (* -> WAIT *)
	SeqEnd_action(N);
END_STEP
TRANSITION FROM SeqEnd TO WaitForStart := TRUE;
END_TRANSITION

ACTION Init_action:
Start:=FALSE;
State:=STATE_WAIT;
MsgOK:=FALSE;
MsgCancel:=FALSE;
SFCRun:=FALSE;
Result:=RESULT_NON;
END_ACTION

ACTION WaitForStart_entry:
;
END_ACTION

ACTION WaitForStart_action:
IF 	Start   THEN
	State:=STATE_RUN;
	Result:=RESULT_NON;
	SFCTimeStart:=TIME();
	Start:=FALSE;
ELSE
	State:=STATE_WAIT;
	MsgOK:=FALSE;
	MsgCancel:=FALSE;
	SFCRun:=FALSE;
END_IF
END_ACTION

ACTION WaitForPart_entry:
ProcessMessage01:='';
Delay.IN:=FALSE;
Delay();
END_ACTION

ACTION WaitForPart_action:
ProcessMessage01:='1IM6';(*warte auf Teil in Vereinzelung*)
Delay.IN:=ST03_461_B69_7.BitInToCheck; 		 (*  ISK anwesend am Stopper *)
Delay.PT:=T#500ms;
Delay();
END_ACTION

ACTION WaitForPart_exit:
ProcessMessage01:='';
END_ACTION

ACTION CloseSeperator_action:
ST03_464_Y71_3.MoveWork:=TRUE;		(* Förderband  Zuführung Vereinzler AST/GST *)
END_ACTION

ACTION OpenStopper_action:
ST03_464_Y71_4.MoveWork:=TRUE;		(* Förderband  Züführung Stopper AST/GST *)
END_ACTION

ACTION WaitForPart__entry:
ProcessMessage01:='';
Delay.IN:=FALSE;
Delay();
END_ACTION

ACTION WaitForPart__action:
ProcessMessage01:='1IM6';(*warte auf Teil in Vereinzelung*)
Delay.IN:=ST03_463_B70_7.BitInToCheck; 		 (* Züführung  ISK auf Übergabeposition Roboter Palettierer  *)
Delay.PT:=T#500ms;
Delay();
END_ACTION

ACTION WaitForPart__exit:
ProcessMessage01:='';
END_ACTION

ACTION CloseStopper_action:
ST03_464_Y71_4.MoveInit:=TRUE;		(*  Förderband  Zuführung Stopper AST/GST*)
END_ACTION

ACTION OpenSeperator_action:
ST03_464_Y71_3.MoveInit:=TRUE;		(* Förderband  Zuführung Vereinzler AST/GST *)
END_ACTION

ACTION SeqEnd_action:
SFCTime:=TIME_TO_DINT(TIME()-SFCTimeStart);
State:=STATE_WAIT;
END_ACTION

TRANSITION AbholPosEmpty:
NOT  ST03_463_B70_7.BitInToCheck
END_TRANSITION

TRANSITION Part Ready:
Delay.Q AND
NOT ST03_463_B70_7.BitInToCheck	AND		(*  Züführung  ISK auf Übergabeposition Roboter Palettierer*)
ST03_461_B69_7.BitInToCheck	AND	(*  ISK anwesend am Vereinzler*)
Robot01.ActualArea <> 4
END_TRANSITION

TRANSITION StateOk:
ST03_464_Y71_3.State=STATE_OK 	(* Förderband  Zuführung Vereinzler AST/GST *)
END_TRANSITION

TRANSITION State Ok:
ST03_464_Y71_4.State=STATE_OK 	(* Förderband  Züführung Stopper AST/GST *)
END_TRANSITION

TRANSITION Part Ready:
Delay.Q AND
Robot01.ActualArea <> 4
END_TRANSITION

TRANSITION State Ok:
ST03_464_Y71_4.State=STATE_OK 	(* Förderband  Züführung Stopper AST/GST *)
END_TRANSITION

TRANSITION StateOk:
ST03_464_Y71_3.State=STATE_OK 	(* Förderband  Zuführung Vereinzler AST/GST *)
END_TRANSITION

TRANSITION WenderDone:
NOT ST03_461_B69_7.BitInToCheck			(*  ISK anwesend am Vereinzler*)
END_TRANSITION
END_PROGRAM

(* POU Stations/ST_03_Ruestsaetze/ST_03_SFCs/Zufuehrungen/ST03_46pol_Wendeeinheit, SFC *)
 PROGRAM ST03_46pol_Wendeeinheit
VAR_OUTPUT
	SFCCurrentPOU			: STRING:='ST03_46pol_Wendeeinheit';
	SFCCurrentStep			: STRING:='';
	FB_CurrentStepHistorie	: FB_CurrentStepHistorie;
	SFCTime					: DINT;
	State   				: StateObject	:= STATE_WAIT;
	Result  				: StateResult;
END_VAR
VAR_INPUT
	Start					:BOOL;
END_VAR
VAR
	MsgOK				: BOOL;
	MsgCancel			: BOOL;
	SFCRun				: BOOL;
	SFCTimeStart		: TIME;
	Delay				: TON;
	(* Userdefinded area *)
	WenderDone			: BOOL;
END_VAR
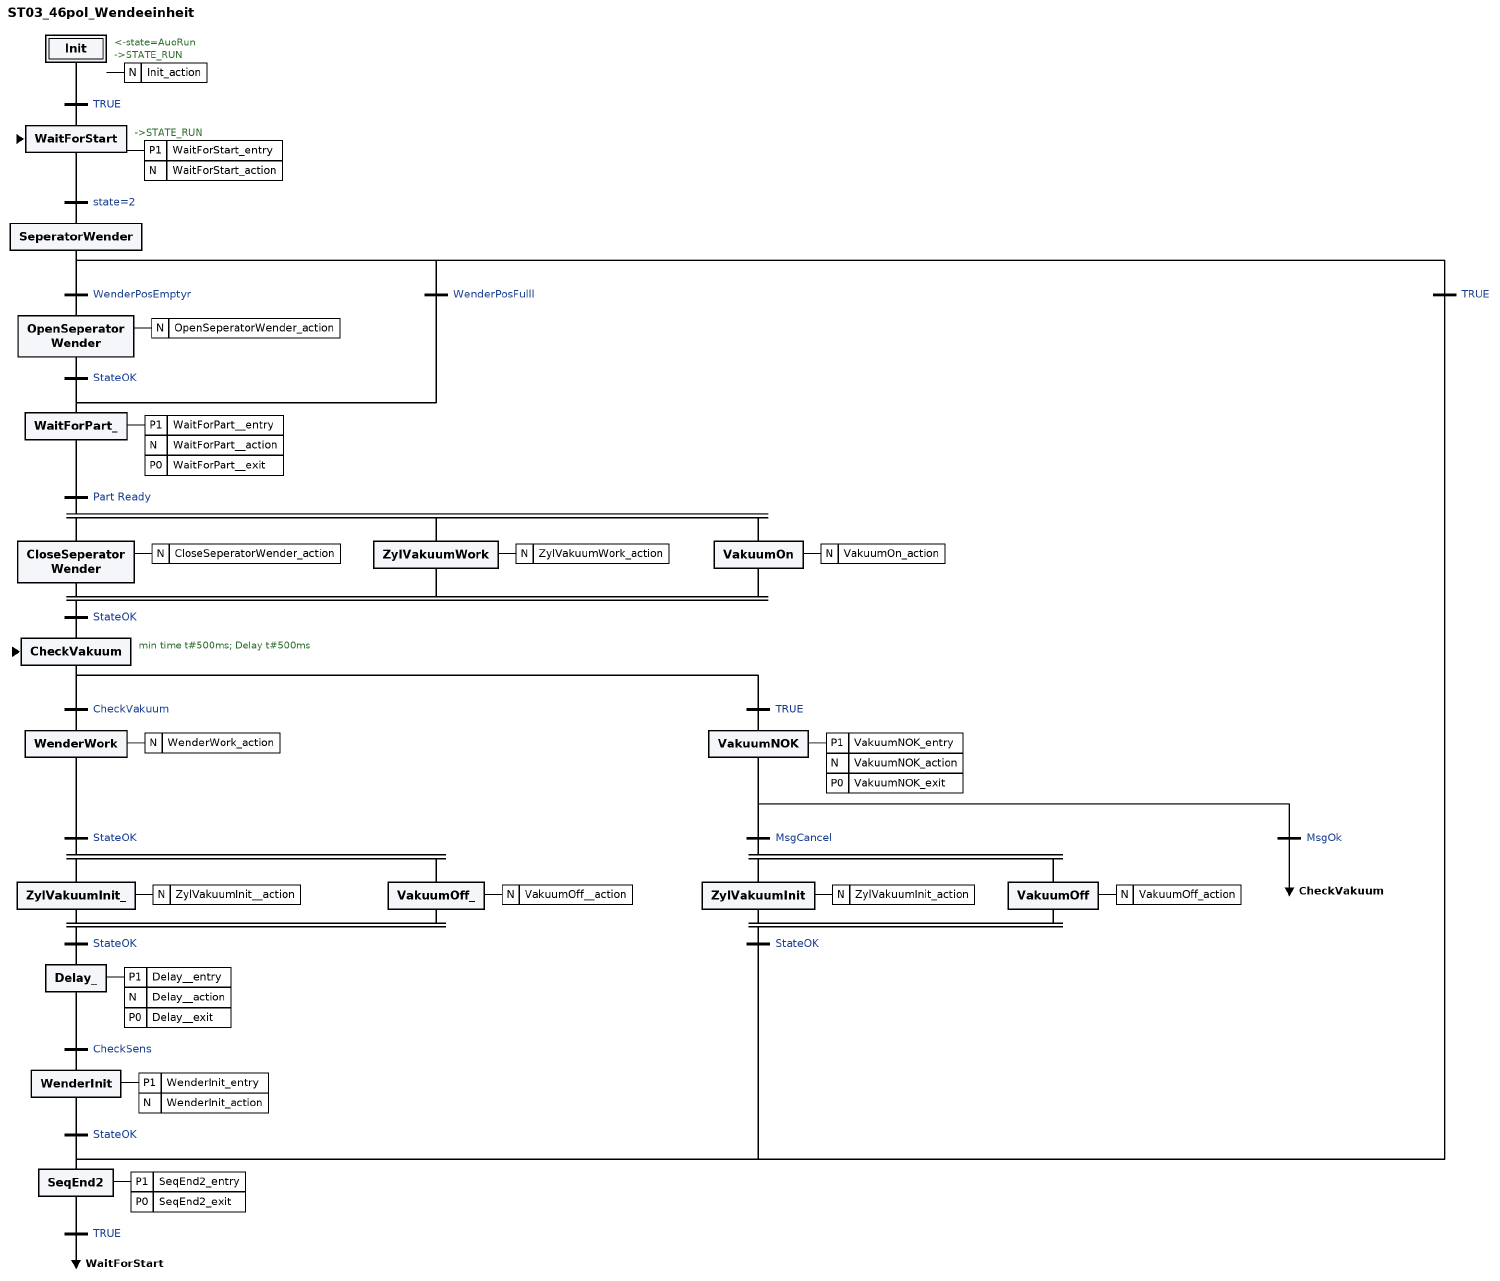
INITIAL_STEP Init: (* <-state=AuoRun / ->STATE_RUN *)
	Init_action(N);
END_STEP
TRANSITION FROM Init TO WaitForStart := TRUE;
END_TRANSITION
STEP WaitForStart: (* ->STATE_RUN *)
	WaitForStart_entry(P1);
	WaitForStart_action(N);
END_STEP
TRANSITION FROM WaitForStart TO SeperatorWender := state=2;
END_TRANSITION
STEP SeperatorWender:
END_STEP
TRANSITION FROM SeperatorWender TO OpenSeperatorWender := WenderPosEmptyr;
END_TRANSITION
TRANSITION FROM SeperatorWender TO WaitForPart_ := WenderPosFulll;
END_TRANSITION
TRANSITION FROM SeperatorWender TO SeqEnd2 := TRUE;
END_TRANSITION
STEP OpenSeperatorWender:
	OpenSeperatorWender_action(N);
END_STEP
TRANSITION FROM OpenSeperatorWender TO WaitForPart_ := StateOK;
END_TRANSITION
STEP WaitForPart_:
	WaitForPart__entry(P1);
	WaitForPart__action(N);
	WaitForPart__exit(P0);
END_STEP
TRANSITION FROM WaitForPart_ TO (CloseSeperatorWender, ZylVakuumWork, VakuumOn) := Part Ready;
END_TRANSITION
STEP CloseSeperatorWender:
	CloseSeperatorWender_action(N);
END_STEP
STEP ZylVakuumWork:
	ZylVakuumWork_action(N);
END_STEP
STEP VakuumOn:
	VakuumOn_action(N);
END_STEP
TRANSITION FROM (CloseSeperatorWender, ZylVakuumWork, VakuumOn) TO CheckVakuum := StateOK;
END_TRANSITION
STEP CheckVakuum: (* min time t#500ms; Delay t#500ms *)
END_STEP
TRANSITION FROM CheckVakuum TO WenderWork := CheckVakuum;
END_TRANSITION
TRANSITION FROM CheckVakuum TO VakuumNOK := TRUE;
END_TRANSITION
STEP WenderWork:
	WenderWork_action(N);
END_STEP
TRANSITION FROM WenderWork TO (ZylVakuumInit_, VakuumOff_) := StateOK;
END_TRANSITION
STEP ZylVakuumInit_:
	ZylVakuumInit__action(N);
END_STEP
STEP VakuumOff_:
	VakuumOff__action(N);
END_STEP
TRANSITION FROM (ZylVakuumInit_, VakuumOff_) TO Delay_ := StateOK;
END_TRANSITION
STEP Delay_:
	Delay__entry(P1);
	Delay__action(N);
	Delay__exit(P0);
END_STEP
TRANSITION FROM Delay_ TO WenderInit := CheckSens;
END_TRANSITION
STEP WenderInit:
	WenderInit_entry(P1);
	WenderInit_action(N);
END_STEP
TRANSITION FROM WenderInit TO SeqEnd2 := StateOK;
END_TRANSITION
STEP VakuumNOK:
	VakuumNOK_entry(P1);
	VakuumNOK_action(N);
	VakuumNOK_exit(P0);
END_STEP
TRANSITION FROM VakuumNOK TO (ZylVakuumInit, VakuumOff) := MsgCancel;
END_TRANSITION
TRANSITION FROM VakuumNOK TO CheckVakuum := MsgOk;
END_TRANSITION
STEP ZylVakuumInit:
	ZylVakuumInit_action(N);
END_STEP
STEP VakuumOff:
	VakuumOff_action(N);
END_STEP
TRANSITION FROM (ZylVakuumInit, VakuumOff) TO SeqEnd2 := StateOK;
END_TRANSITION
STEP SeqEnd2:
	SeqEnd2_entry(P1);
	SeqEnd2_exit(P0);
END_STEP
TRANSITION FROM SeqEnd2 TO WaitForStart := TRUE;
END_TRANSITION

ACTION Init_action:
Start:=FALSE;
State:=STATE_WAIT;
MsgOK:=FALSE;
MsgCancel:=FALSE;
SFCRun:=FALSE;
Result:=RESULT_NON;
END_ACTION

ACTION WaitForStart_entry:
;
END_ACTION

ACTION WaitForStart_action:
IF 	Start   THEN
	State:=STATE_RUN;
	Result:=RESULT_NON;
	SFCTimeStart:=TIME();
	Start:=FALSE;
	WenderDone:=FALSE;
ELSE
	State:=STATE_WAIT;
	MsgOK:=FALSE;
	MsgCancel:=FALSE;
	SFCRun:=FALSE;
END_IF
END_ACTION

ACTION OpenSeperatorWender_action:
ST03_464_Y71_0.MoveInit:=TRUE;		(* Förderband  Zuführung Vereinzelner Wender AST/GST *)
END_ACTION

ACTION WaitForPart__entry:
ProcessMessage01:='';
Delay.IN:=FALSE;
Delay();
END_ACTION

ACTION WaitForPart__action:
ProcessMessage01:='1IM6';(*'warte auf Teil in Vereinzelung*)
Delay.IN:=ST03_462_B70_0.BitInToCheck; 		 (* Züführung  ISK auf Übergabeposition Roboter Palettierer  *)
Delay.PT:=T#800ms;
Delay();
END_ACTION

ACTION WaitForPart__exit:
ProcessMessage01:='';
END_ACTION

ACTION CloseSeperatorWender_action:
ST03_464_Y71_0.MoveWork:=TRUE;		(* Förderband  Zuführung Vereinzelner Wender AST/GST *)
END_ACTION

ACTION ZylVakuumWork_action:
ST03_464_Y71_1.MoveWork:=TRUE;		(*  Förderband  Zuführung Zylinder Vakuumdüsen AST/GST*)
END_ACTION

ACTION VakuumOn_action:
ST03_464_Y71_5.MoveWork:=TRUE;	(*  Förderband  Vakuumdüsen EIN/AUS *)
END_ACTION

ACTION WenderWork_action:
ST03_464_Y71_2.MoveWork:=TRUE;		(* Förderband  Zuführung Wender Einlauf / Auslauf *)
END_ACTION

ACTION ZylVakuumInit__action:
ST03_464_Y71_1.MoveInit:=TRUE;		(*  Förderband  Zuführung Zylinder Vakuumdüsen AST/GST*)
END_ACTION

ACTION VakuumOff__action:
ST03_464_Y71_5.MoveInit:=TRUE;	(*  Förderband  Vakuumdüsen EIN/AUS *)
END_ACTION

ACTION Delay__entry:
Delay(IN:=FALSE);
END_ACTION

ACTION Delay__action:
Delay(IN:=TRUE,PT:=t#2000ms);
END_ACTION

ACTION Delay__exit:
Delay(IN:=FALSE);
END_ACTION

ACTION WenderInit_entry:
Delay(IN:=FALSE);
END_ACTION

ACTION WenderInit_action:
ST03_464_Y71_2.MoveInit:=TRUE;		(* Förderband  Zuführung Wender Einlauf / Auslauf *)
END_ACTION

ACTION VakuumNOK_entry:
MessageHandler.ClearMessageLines(sVisu:=Visu.Message);
END_ACTION

ACTION VakuumNOK_action:
MessageHandler.Msg.ID:='PM119';
MessageHandler.Msg.Name:='Vakuum nicht OK';
MessageHandler.Msg.Text:='ST03 Vakuum an der Wendestation nicht OK';
MessageHandler.Msg.Color:=Color.red;
MessageHandler.Msg.Station:=1;


MessageHandler(
	Prio:=2, 							(*1=highest, .. , 4=lowest*)
	Btn1Addr:=ADR(MsgOk),			(*Address of Button1 , if Zero then Button is unvisible*)
	Btn2Addr:=ADR(MsgCancel),			(*Address of Button2 , if Zero then Button is unvisible*)
	sVisu:=Visu.Message);
END_ACTION

ACTION VakuumNOK_exit:
MsgOk:=FALSE;
MsgCancel:=FALSE;
END_ACTION

ACTION ZylVakuumInit_action:
ST03_464_Y71_1.MoveInit:=TRUE;		(*  Förderband  Zuführung Zylinder Vakuumdüsen AST/GST*)
END_ACTION

ACTION VakuumOff_action:
ST03_464_Y71_5.MoveInit:=TRUE;	(*  Förderband  Vakuumdüsen EIN/AUS *)
END_ACTION

ACTION SeqEnd2_entry:
WenderDone:=TRUE;
END_ACTION

ACTION SeqEnd2_exit:
WenderDone:=FALSE;
END_ACTION

TRANSITION WenderPosEmptyr:
NOT ST03_462_B70_0.BitInToCheck AND	(*Förderband  ISK anwesend Wender*)
NOT  ST03_464_B71_7.BitInToCheck	 AND	(*Förderband   Staustrecke mitte voll*)
ST03_463_B70_5.ValveSensor				(* Züführung  ISK Wendestation Einlauf GST*)
END_TRANSITION

TRANSITION StateOK:
ST03_464_Y71_0.State = STATE_OK 	(* Förderband  Zuführung Vereinzelner Wender AST/GST *)
END_TRANSITION

TRANSITION WenderPosFulll:
ST03_462_B70_0.BitInToCheck AND	(*Förderband  ISK anwesend Wender*)
NOT  ST03_464_B71_7.BitInToCheck  AND	(*Förderband   Staustrecke mitte voll*)
ST03_463_B70_5.ValveSensor				(* Züführung  ISK Wendestation Einlauf GST*)
END_TRANSITION

TRANSITION Part Ready:
Delay.Q
END_TRANSITION

TRANSITION StateOK:
ST03_464_Y71_0.State = STATE_OK AND	(* Förderband  Zuführung Vereinzelner Wender AST/GST *)
ST03_464_Y71_1.State = STATE_OK	AND	(*   Förderband  Zuführung Zylinder Vakuumdüsen AST/GST *)
ST03_464_Y71_5.State = STATE_OK		(*  Förderband  Vakuumdüsen EIN/AUS *)
END_TRANSITION

TRANSITION CheckVakuum:
ST03_464_B71_6.BitInToCheck	(*Förderband  Vakuum vorhanden*)
END_TRANSITION

TRANSITION StateOK:
ST03_464_Y71_2.State = STATE_OK 	(* Förderband  ZuführungWender Einlauf / Auslauf  *)
END_TRANSITION

TRANSITION StateOK:
ST03_464_Y71_1.State = STATE_OK	AND	(*   Förderband  Zuführung Zylinder Vakuumdüsen AST/GST *)
ST03_464_Y71_5.State = STATE_OK		(*  Förderband  Vakuumdüsen EIN/AUS *)
END_TRANSITION

TRANSITION CheckSens:
ST03_464_B71_7.BitInToCheck	(* Förderband   Staustrecke mitte vol*) OR
delay.Q
END_TRANSITION

TRANSITION StateOK:
ST03_464_Y71_2.State = STATE_OK 	(* Förderband  ZuführungWender Einlauf / Auslauf  *)
END_TRANSITION

TRANSITION StateOK:
ST03_464_Y71_1.State = STATE_OK	AND	(*   Förderband  Zuführung Zylinder Vakuumdüsen AST/GST *)
ST03_464_Y71_5.State = STATE_OK		(*  Förderband  Vakuumdüsen EIN/AUS *)
END_TRANSITION
END_PROGRAM

(* POU Stations/ST_03_Ruestsaetze/ST_03_SFCs/Zufuehrungen/ST03_NOX_4pol_Zufuehrung, SFC *)
 PROGRAM ST03_NOX_4pol_Zufuehrung
VAR_OUTPUT
	SFCCurrentPOU		: STRING:='ST03_NOX_4pol_Zufuehrung';
	SFCCurrentStep		: STRING:='';
	FB_CurrentStepHistorie:FB_CurrentStepHistorie;
	SFCTime			: DINT;
	State   				: StateObject	:= STATE_WAIT;
	Result  				: StateResult;
END_VAR
VAR_INPUT
	Start					:BOOL;
END_VAR
VAR
	MsgOK				: BOOL;
	MsgCancel			: BOOL;
	SFCRun				: BOOL;
	SFCTimeStart		: TIME;
	Delay				: TON;
	(* Userdefinded area *)

END_VAR
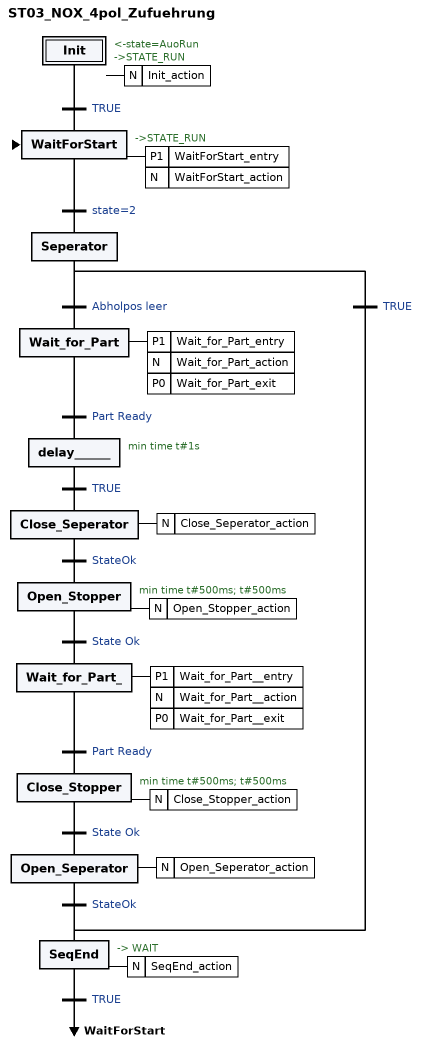
INITIAL_STEP Init: (* <-state=AuoRun / ->STATE_RUN *)
	Init_action(N);
END_STEP
TRANSITION FROM Init TO WaitForStart := TRUE;
END_TRANSITION
STEP WaitForStart: (* ->STATE_RUN *)
	WaitForStart_entry(P1);
	WaitForStart_action(N);
END_STEP
TRANSITION FROM WaitForStart TO Seperator := state=2;
END_TRANSITION
STEP Seperator:
END_STEP
TRANSITION FROM Seperator TO Wait_for_Part := Abholpos leer;
END_TRANSITION
TRANSITION FROM Seperator TO SeqEnd := TRUE;
END_TRANSITION
STEP Wait_for_Part:
	Wait_for_Part_entry(P1);
	Wait_for_Part_action(N);
	Wait_for_Part_exit(P0);
END_STEP
TRANSITION FROM Wait_for_Part TO delay______ := Part Ready;
END_TRANSITION
STEP delay______: (* min time t#1s *)
END_STEP
TRANSITION FROM delay______ TO Close_Seperator := TRUE;
END_TRANSITION
STEP Close_Seperator:
	Close_Seperator_action(N);
END_STEP
TRANSITION FROM Close_Seperator TO Open_Stopper := StateOk;
END_TRANSITION
STEP Open_Stopper: (* min time t#500ms; t#500ms *)
	Open_Stopper_action(N);
END_STEP
TRANSITION FROM Open_Stopper TO Wait_for_Part_ := State Ok;
END_TRANSITION
STEP Wait_for_Part_:
	Wait_for_Part__entry(P1);
	Wait_for_Part__action(N);
	Wait_for_Part__exit(P0);
END_STEP
TRANSITION FROM Wait_for_Part_ TO Close_Stopper := Part Ready;
END_TRANSITION
STEP Close_Stopper: (* min time t#500ms; t#500ms *)
	Close_Stopper_action(N);
END_STEP
TRANSITION FROM Close_Stopper TO Open_Seperator := State Ok;
END_TRANSITION
STEP Open_Seperator:
	Open_Seperator_action(N);
END_STEP
TRANSITION FROM Open_Seperator TO SeqEnd := StateOk;
END_TRANSITION
STEP SeqEnd: (* -> WAIT *)
	SeqEnd_action(N);
END_STEP
TRANSITION FROM SeqEnd TO WaitForStart := TRUE;
END_TRANSITION

ACTION Init_action:
Start:=FALSE;
State:=STATE_WAIT;
MsgOK:=FALSE;
MsgCancel:=FALSE;
SFCRun:=FALSE;
Result:=RESULT_NON;
END_ACTION

ACTION WaitForStart_entry:
;
END_ACTION

ACTION WaitForStart_action:
IF 	Start   THEN
	State:=STATE_RUN;
	Result:=RESULT_NON;
	SFCTimeStart:=TIME();
	Start:=FALSE;
ELSE
	State:=STATE_WAIT;
	MsgOK:=FALSE;
	MsgCancel:=FALSE;
	SFCRun:=FALSE;
END_IF
END_ACTION

ACTION Wait_for_Part_entry:
ProcessMessage01:='';
Delay.IN:=FALSE;
Delay();
END_ACTION

ACTION Wait_for_Part_action:
ProcessMessage01:='1IM9';(*warte auf Teil in Stopper*)
Delay.IN:=ST03_491_B69_5.BitInToCheck; 		(*  ISK an stopper.*)
Delay.PT:=T#500ms;
Delay();
END_ACTION

ACTION Wait_for_Part_exit:
ProcessMessage01:='';
END_ACTION

ACTION Close_Seperator_action:
ST03_492_Y70_0.MoveWork:=TRUE;		(* Förderband  Zuführung Vereinzler AST/GST *)
END_ACTION

ACTION Open_Stopper_action:
ST03_492_Y70_1.MoveWork:=TRUE;		(* Förderband  Züführung Stopper AST/GST *)
END_ACTION

ACTION Wait_for_Part__entry:
ProcessMessage01:='';
Delay.IN:=FALSE;
Delay();
END_ACTION

ACTION Wait_for_Part__action:
ProcessMessage01:='1IM10';(*warte auf Teil in Abholposition*)
Delay.IN:=ST03_491_B69_7.BitInToCheck; 		 (* Schnittstelle Iso auf Übergabeposition Roboter *)
Delay.PT:=T#500ms;
Delay();
END_ACTION

ACTION Wait_for_Part__exit:
ProcessMessage01:='';
END_ACTION

ACTION Close_Stopper_action:
ST03_492_Y70_1.MoveInit:=TRUE;		(* Förderband  Züführung Stopper AST/GST *)
END_ACTION

ACTION Open_Seperator_action:
ST03_492_Y70_0.MoveInit:=TRUE;		(* Förderband  Zuführung Vereinzler AST/GST *)
END_ACTION

ACTION SeqEnd_action:
SFCTime:=TIME_TO_DINT(TIME()-SFCTimeStart);
State:=STATE_WAIT;
END_ACTION

TRANSITION Abholpos leer:
NOT  ST03_491_B69_7.BitInToCheck		(*  ISK auf Abholposition Robi*)
END_TRANSITION

TRANSITION Part Ready:
Delay.Q AND
NOT ST03_491_B69_7.BitInToCheck	AND		(*  ISK auf Abholposition Robi*)
ST03_491_B69_5.BitInToCheck	AND				(*  ISK anwesend am Stoper*)
Robot01.ActualArea <> 4
END_TRANSITION

TRANSITION StateOk:
ST03_492_Y70_0.State=STATE_OK 	(* Förderband  Zuführung Vereinzler AST/GST *)
END_TRANSITION

TRANSITION State Ok:
ST03_492_Y70_1.State=STATE_OK 	(* Förderband  Züführung Stopper AST/GST *)
END_TRANSITION

TRANSITION Part Ready:
Delay.Q AND
Robot01.ActualArea <> 4
END_TRANSITION

TRANSITION State Ok:
ST03_492_Y70_1.State=STATE_OK 	(* Förderband  Züführung Stopper AST/GST *)
END_TRANSITION

TRANSITION StateOk:
ST03_492_Y70_0.State=STATE_OK 	(* Förderband  Zuführung Vereinzler AST/GST *)
END_TRANSITION
END_PROGRAM

(* POU Stations/ST_03_Ruestsaetze/ST_03_SFCs/Zufuehrungen/ST03_88pol_Zufuehrung, SFC *)
 PROGRAM ST03_88pol_Zufuehrung
VAR_OUTPUT
	SFCCurrentPOU			: STRING:='ST03_88pol_Zufuehrung';
	SFCCurrentStep			: STRING:='';
	FB_CurrentStepHistorie:FB_CurrentStepHistorie;
	SFCTime					: DINT;
	State   				: StateObject	:= STATE_WAIT;
	Result  				: StateResult;
END_VAR
VAR_INPUT
	Start					:BOOL;
END_VAR
VAR
	MsgOK				: BOOL;
	MsgCancel			: BOOL;
	SFCRun				: BOOL;
	SFCTimeStart		: TIME;
	Delay				: TON;
	(* Userdefinded area *)

END_VAR
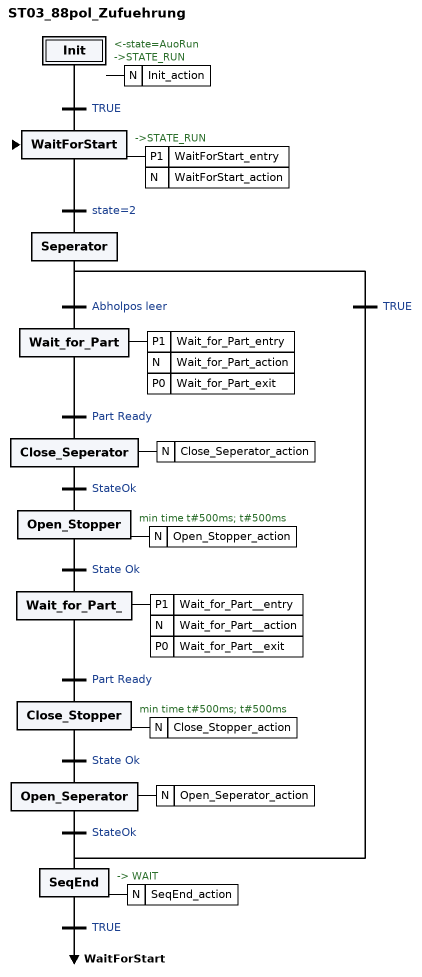
INITIAL_STEP Init: (* <-state=AuoRun / ->STATE_RUN *)
	Init_action(N);
END_STEP
TRANSITION FROM Init TO WaitForStart := TRUE;
END_TRANSITION
STEP WaitForStart: (* ->STATE_RUN *)
	WaitForStart_entry(P1);
	WaitForStart_action(N);
END_STEP
TRANSITION FROM WaitForStart TO Seperator := state=2;
END_TRANSITION
STEP Seperator:
END_STEP
TRANSITION FROM Seperator TO Wait_for_Part := Abholpos leer;
END_TRANSITION
TRANSITION FROM Seperator TO SeqEnd := TRUE;
END_TRANSITION
STEP Wait_for_Part:
	Wait_for_Part_entry(P1);
	Wait_for_Part_action(N);
	Wait_for_Part_exit(P0);
END_STEP
TRANSITION FROM Wait_for_Part TO Close_Seperator := Part Ready;
END_TRANSITION
STEP Close_Seperator:
	Close_Seperator_action(N);
END_STEP
TRANSITION FROM Close_Seperator TO Open_Stopper := StateOk;
END_TRANSITION
STEP Open_Stopper: (* min time t#500ms; t#500ms *)
	Open_Stopper_action(N);
END_STEP
TRANSITION FROM Open_Stopper TO Wait_for_Part_ := State Ok;
END_TRANSITION
STEP Wait_for_Part_:
	Wait_for_Part__entry(P1);
	Wait_for_Part__action(N);
	Wait_for_Part__exit(P0);
END_STEP
TRANSITION FROM Wait_for_Part_ TO Close_Stopper := Part Ready;
END_TRANSITION
STEP Close_Stopper: (* min time t#500ms; t#500ms *)
	Close_Stopper_action(N);
END_STEP
TRANSITION FROM Close_Stopper TO Open_Seperator := State Ok;
END_TRANSITION
STEP Open_Seperator:
	Open_Seperator_action(N);
END_STEP
TRANSITION FROM Open_Seperator TO SeqEnd := StateOk;
END_TRANSITION
STEP SeqEnd: (* -> WAIT *)
	SeqEnd_action(N);
END_STEP
TRANSITION FROM SeqEnd TO WaitForStart := TRUE;
END_TRANSITION

ACTION Init_action:
Start:=FALSE;
State:=STATE_WAIT;
MsgOK:=FALSE;
MsgCancel:=FALSE;
SFCRun:=FALSE;
Result:=RESULT_NON;
END_ACTION

ACTION WaitForStart_entry:
State:=STATE_OK;
END_ACTION

ACTION WaitForStart_action:
IF 	Start   THEN
	State:=STATE_RUN;
	Result:=RESULT_NON;
	SFCTimeStart:=TIME();
	Start:=FALSE;
ELSE
	State:=STATE_WAIT;
	MsgOK:=FALSE;
	MsgCancel:=FALSE;
	SFCRun:=FALSE;
END_IF
END_ACTION

ACTION Wait_for_Part_entry:
ProcessMessage01:='';
Delay.IN:=FALSE;
Delay();
END_ACTION

ACTION Wait_for_Part_action:
State:=STATE_RUN;
ProcessMessage01:='1IM9';(*warte auf Teil in Stopper*)
Delay.IN:=ST03_501_B69_6.BitInToCheck; 		(*  ISK an stopper.*)
Delay.PT:=T#500ms;
Delay();
END_ACTION

ACTION Wait_for_Part_exit:
ProcessMessage01:='';
END_ACTION

ACTION Close_Seperator_action:
ST03_502_Y70_1.MoveWork:=TRUE;		(* Förderband  Zuführung Vereinzler AST/GST *)
END_ACTION

ACTION Open_Stopper_action:
ST03_502_Y70_2.MoveWork:=TRUE;		(* Förderband  Züführung Stopper AST/GST *)
END_ACTION

ACTION Wait_for_Part__entry:
ProcessMessage01:='';
Delay.IN:=FALSE;
Delay();
END_ACTION

ACTION Wait_for_Part__action:
ProcessMessage01:='1IM10';(*warte auf Teil in Abholposition*)
Delay.IN:=ST03_501_B69_7.BitInToCheck; 		 (* ISK auf Abholposition Robi *)
Delay.PT:=T#500ms;
Delay();
END_ACTION

ACTION Wait_for_Part__exit:
ProcessMessage01:='';
END_ACTION

ACTION Close_Stopper_action:
ST03_502_Y70_2.MoveInit:=TRUE;		(* Förderband  Züführung Stopper AST/GST *)
END_ACTION

ACTION Open_Seperator_action:
ST03_502_Y70_1.MoveInit:=TRUE;		(* Förderband  Zuführung Vereinzler AST/GST *)
END_ACTION

ACTION SeqEnd_action:
SFCTime:=TIME_TO_DINT(TIME()-SFCTimeStart);
State:=STATE_WAIT;
END_ACTION

TRANSITION Abholpos leer:
NOT  ST03_501_B69_7.BitInToCheck		(*  ISK auf Abholposition Robi*)
END_TRANSITION

TRANSITION Part Ready:
Delay.Q AND
NOT ST03_501_B69_7.BitInToCheck	AND		(*  ISK auf Abholposition Robi*)
ST03_501_B69_6.BitInToCheck	AND				(*  ISK anwesend am Stoper*)
Robot01.ActualArea <> 4
END_TRANSITION

TRANSITION StateOk:
ST03_502_Y70_1.State=STATE_OK 	(* Förderband  Zuführung Vereinzler AST/GST *)
END_TRANSITION

TRANSITION State Ok:
ST03_502_Y70_2.State=STATE_OK 	(* Förderband  Züführung Stopper AST/GST *)
END_TRANSITION

TRANSITION Part Ready:
Delay.Q AND
Robot01.ActualArea <> 4
END_TRANSITION

TRANSITION State Ok:
ST03_502_Y70_2.State=STATE_OK 	(* Förderband  Züführung Stopper AST/GST *)
END_TRANSITION

TRANSITION StateOk:
ST03_502_Y70_1.State=STATE_OK 	(* Förderband  Zuführung Vereinzler AST/GST *)
END_TRANSITION
END_PROGRAM

(* POU Stations/ST_03_Ruestsaetze/ST_03_SFCs/Zufuehrungen/ST03_7pol_Zufuehrung, SFC *)
 PROGRAM ST03_7pol_Zufuehrung
VAR_OUTPUT
	SFCCurrentPOU			: STRING:='ST03_7pol_Zufuehrung';
	SFCCurrentStep			: STRING:='';
	FB_CurrentStepHistorie	:FB_CurrentStepHistorie;
	SFCTime					: DINT;
	State   				: StateObject	:= STATE_WAIT;
	Result  				: StateResult;
END_VAR
VAR_INPUT
	Start					:BOOL;
END_VAR
VAR
	MsgOK				: BOOL;
	MsgCancel			: BOOL;
	SFCRun			: BOOL;
	SFCTimeStart		: TIME;
	Delay				: TON;
	Delay2				: TON;
	(* Userdefinded area *)

END_VAR
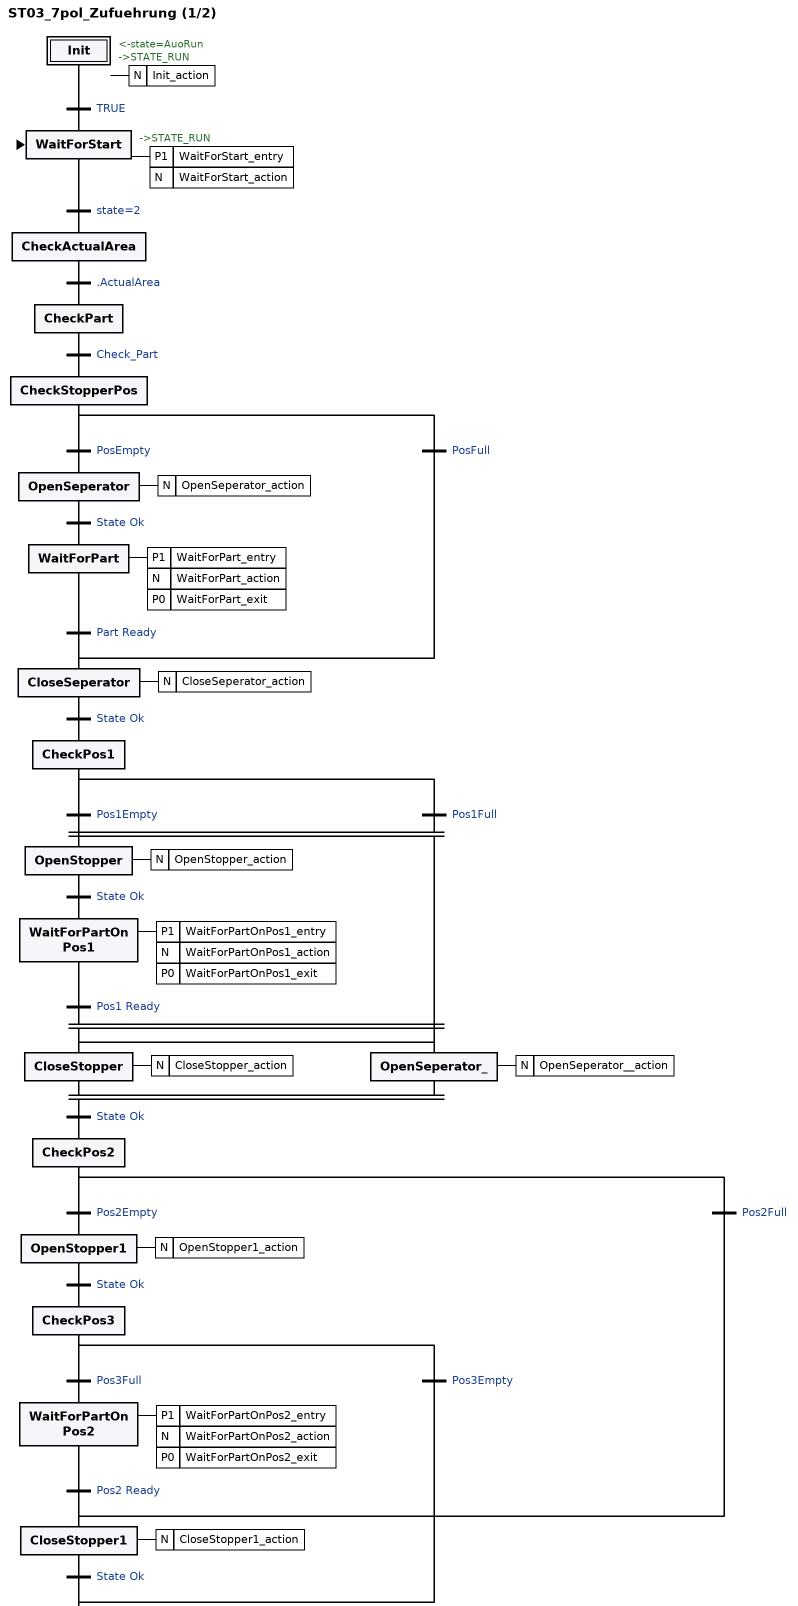
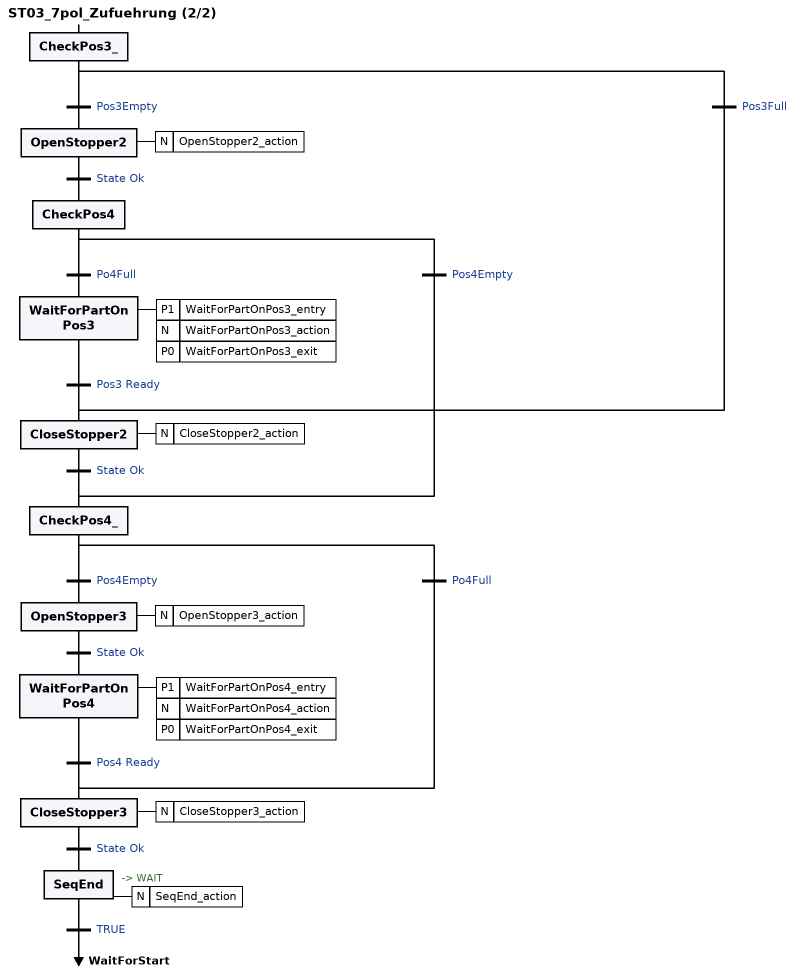
INITIAL_STEP Init: (* <-state=AuoRun / ->STATE_RUN *)
	Init_action(N);
END_STEP
TRANSITION FROM Init TO WaitForStart := TRUE;
END_TRANSITION
STEP WaitForStart: (* ->STATE_RUN *)
	WaitForStart_entry(P1);
	WaitForStart_action(N);
END_STEP
TRANSITION FROM WaitForStart TO CheckActualArea  := state=2;
END_TRANSITION
STEP CheckActualArea :
END_STEP
TRANSITION FROM CheckActualArea  TO CheckPart := .ActualArea;
END_TRANSITION
STEP CheckPart:
END_STEP
TRANSITION FROM CheckPart TO CheckStopperPos := Check_Part;
END_TRANSITION
STEP CheckStopperPos:
END_STEP
TRANSITION FROM CheckStopperPos TO OpenSeperator := PosEmpty;
END_TRANSITION
TRANSITION FROM CheckStopperPos TO CloseSeperator := PosFull;
END_TRANSITION
STEP OpenSeperator:
	OpenSeperator_action(N);
END_STEP
TRANSITION FROM OpenSeperator TO WaitForPart := State Ok;
END_TRANSITION
STEP WaitForPart:
	WaitForPart_entry(P1);
	WaitForPart_action(N);
	WaitForPart_exit(P0);
END_STEP
TRANSITION FROM WaitForPart TO CloseSeperator := Part Ready;
END_TRANSITION
STEP CloseSeperator:
	CloseSeperator_action(N);
END_STEP
TRANSITION FROM CloseSeperator TO CheckPos1 := State Ok;
END_TRANSITION
STEP CheckPos1:
END_STEP
TRANSITION FROM CheckPos1 TO OpenStopper := Pos1Empty;
END_TRANSITION
TRANSITION FROM CheckPos1 TO (CloseStopper, OpenSeperator_) := Pos1Full;
END_TRANSITION
STEP OpenStopper:
	OpenStopper_action(N);
END_STEP
TRANSITION FROM OpenStopper TO WaitForPartOnPos1 := State Ok;
END_TRANSITION
STEP WaitForPartOnPos1:
	WaitForPartOnPos1_entry(P1);
	WaitForPartOnPos1_action(N);
	WaitForPartOnPos1_exit(P0);
END_STEP
TRANSITION FROM WaitForPartOnPos1 TO (CloseStopper, OpenSeperator_) := Pos1 Ready;
END_TRANSITION
STEP CloseStopper:
	CloseStopper_action(N);
END_STEP
STEP OpenSeperator_:
	OpenSeperator__action(N);
END_STEP
TRANSITION FROM (CloseStopper, OpenSeperator_) TO CheckPos2 := State Ok;
END_TRANSITION
STEP CheckPos2:
END_STEP
TRANSITION FROM CheckPos2 TO OpenStopper1 := Pos2Empty;
END_TRANSITION
TRANSITION FROM CheckPos2 TO CloseStopper1 := Pos2Full;
END_TRANSITION
STEP OpenStopper1:
	OpenStopper1_action(N);
END_STEP
TRANSITION FROM OpenStopper1 TO CheckPos3 := State Ok;
END_TRANSITION
STEP CheckPos3:
END_STEP
TRANSITION FROM CheckPos3 TO WaitForPartOnPos2 := Pos3Full;
END_TRANSITION
TRANSITION FROM CheckPos3 TO CheckPos3_ := Pos3Empty;
END_TRANSITION
STEP WaitForPartOnPos2:
	WaitForPartOnPos2_entry(P1);
	WaitForPartOnPos2_action(N);
	WaitForPartOnPos2_exit(P0);
END_STEP
TRANSITION FROM WaitForPartOnPos2 TO CloseStopper1 := Pos2 Ready;
END_TRANSITION
STEP CloseStopper1:
	CloseStopper1_action(N);
END_STEP
TRANSITION FROM CloseStopper1 TO CheckPos3_ := State Ok;
END_TRANSITION
STEP CheckPos3_:
END_STEP
TRANSITION FROM CheckPos3_ TO OpenStopper2 := Pos3Empty;
END_TRANSITION
TRANSITION FROM CheckPos3_ TO CloseStopper2 := Pos3Full;
END_TRANSITION
STEP OpenStopper2:
	OpenStopper2_action(N);
END_STEP
TRANSITION FROM OpenStopper2 TO CheckPos4 := State Ok;
END_TRANSITION
STEP CheckPos4:
END_STEP
TRANSITION FROM CheckPos4 TO WaitForPartOnPos3 := Po4Full;
END_TRANSITION
TRANSITION FROM CheckPos4 TO CheckPos4_ := Pos4Empty;
END_TRANSITION
STEP WaitForPartOnPos3:
	WaitForPartOnPos3_entry(P1);
	WaitForPartOnPos3_action(N);
	WaitForPartOnPos3_exit(P0);
END_STEP
TRANSITION FROM WaitForPartOnPos3 TO CloseStopper2 := Pos3 Ready;
END_TRANSITION
STEP CloseStopper2:
	CloseStopper2_action(N);
END_STEP
TRANSITION FROM CloseStopper2 TO CheckPos4_ := State Ok;
END_TRANSITION
STEP CheckPos4_:
END_STEP
TRANSITION FROM CheckPos4_ TO OpenStopper3 := Pos4Empty;
END_TRANSITION
TRANSITION FROM CheckPos4_ TO CloseStopper3 := Po4Full;
END_TRANSITION
STEP OpenStopper3:
	OpenStopper3_action(N);
END_STEP
TRANSITION FROM OpenStopper3 TO WaitForPartOnPos4 := State Ok;
END_TRANSITION
STEP WaitForPartOnPos4:
	WaitForPartOnPos4_entry(P1);
	WaitForPartOnPos4_action(N);
	WaitForPartOnPos4_exit(P0);
END_STEP
TRANSITION FROM WaitForPartOnPos4 TO CloseStopper3 := Pos4 Ready;
END_TRANSITION
STEP CloseStopper3:
	CloseStopper3_action(N);
END_STEP
TRANSITION FROM CloseStopper3 TO SeqEnd := State Ok;
END_TRANSITION
STEP SeqEnd: (* -> WAIT *)
	SeqEnd_action(N);
END_STEP
TRANSITION FROM SeqEnd TO WaitForStart := TRUE;
END_TRANSITION

ACTION Init_action:
Start:=FALSE;
State:=STATE_WAIT;
MsgOK:=FALSE;
MsgCancel:=FALSE;
SFCRun:=FALSE;
Result:=RESULT_NON;
END_ACTION

ACTION WaitForStart_entry:
;
END_ACTION

ACTION WaitForStart_action:
IF 	Start   THEN
	State:=STATE_RUN;
	Result:=RESULT_NON;
	SFCTimeStart:=TIME();
	Start:=FALSE;
ELSE
	State:=STATE_WAIT;
	MsgOK:=FALSE;
	MsgCancel:=FALSE;
	SFCRun:=FALSE;
END_IF
END_ACTION

ACTION OpenSeperator_action:
ST03_515_Y72_2.MoveInit:=TRUE;		(* Führungsschiene  Zuführung Vereinzler AST/GST *)
END_ACTION

ACTION WaitForPart_entry:
ProcessMessage02:='';
Delay(IN:=FALSE);
END_ACTION

ACTION WaitForPart_action:
ProcessMessage02:='2IM6';						(*warte auf Teil Übergabeposition 1*)
END_ACTION

ACTION WaitForPart_exit:
ProcessMessage02:='';
END_ACTION

ACTION CloseSeperator_action:
ST03_515_Y72_2.MoveWork:=TRUE;		(* Führungsschiene  Zuführung Vereinzler AST/GST *)
END_ACTION

ACTION OpenStopper_action:
ST03_515_Y72_3.MoveWork:=TRUE;		(* Führungsschiene  Zuführung Stopper AST/GST *)
END_ACTION

ACTION WaitForPartOnPos1_entry:
ProcessMessage02:='';
Delay(IN:=FALSE);
END_ACTION

ACTION WaitForPartOnPos1_action:
ProcessMessage02:='2IM6';						(*warte auf Teil Übergabeposition 1*)
END_ACTION

ACTION WaitForPartOnPos1_exit:
ProcessMessage02:='';
END_ACTION

ACTION CloseStopper_action:
ST03_515_Y72_3.MoveInit:=TRUE;		(* Führungsschiene  Zuführung Stopper AST/GST *)
END_ACTION

ACTION OpenSeperator__action:
ST03_515_Y72_2.MoveInit:=TRUE;		(* Führungsschiene  Zuführung Vereinzler AST/GST *)
END_ACTION

ACTION OpenStopper1_action:
ST03_515_Y72_4.MoveWork:=TRUE;		(* Übergabeposition Stopper 1 *)
END_ACTION

ACTION WaitForPartOnPos2_entry:
ProcessMessage02:='';
Delay(IN:=FALSE);
END_ACTION

ACTION WaitForPartOnPos2_action:
ProcessMessage02:='2IM5';						(*warte auf Teil Übergabeposition 2*)
END_ACTION

ACTION WaitForPartOnPos2_exit:
ProcessMessage02:='';
END_ACTION

ACTION CloseStopper1_action:
ST03_515_Y72_4.MoveInit:=TRUE;		(* Übergabeposition Stopper 1 *)
END_ACTION

